LIN {X 0,Y 516.88,Z 308.725,A -85,B 0,C 180,E1 -5018.462,E2 -5018.462} C_VEL
LIN {X 0,Y 516.899,Z 308.722,A -85,B 0,C 180,E1 -5020.954,E2 -5020.954} C_VEL
LIN {X 0,Y 516.911,Z 308.717,A -85,B 0,C 180,E1 -5023.41,E2 -5023.41} C_VEL
LIN {X 0,Y 516.889,Z 308.719,A -85,B 0,C 180,E1 -5025.833,E2 -5025.833} C_VEL
LIN {X 0,Y 516.958,Z 308.715,A -85,B 0,C 180,E1 -5028.233,E2 -5028.233} C_VEL
LIN {X 0,Y 516.963,Z 308.71,A -85,B 0,C 180,E1 -5031.399,E2 -5031.399} C_VEL
LIN {X 0,Y 517.004,Z 308.705,A -85,B 0,C 180,E1 -5033.757,E2 -5033.757} C_VEL
LIN {X 0,Y 517.078,Z 308.696,A -85,B 0,C 180,E1 -5037.663,E2 -5037.663} C_VEL
LIN {X 0,Y 517.088,Z 308.697,A -85,B 0,C 180,E1 -5040.779,E2 -5040.779} C_VEL
LIN {X 0,Y 517.009,Z 308.704,A -85,B 0,C 180,E1 -5043.117,E2 -5043.117} C_VEL
LIN {X 0,Y 517.003,Z 308.713,A -85,B 0,C 180,E1 -5046.243,E2 -5046.243} C_VEL
LIN {X 0,Y 516.948,Z 308.712,A -85,B 0,C 180,E1 -5049.389,E2 -5049.389} C_VEL
LIN {X 0,Y 516.975,Z 308.712,A -85,B 0,C 180,E1 -5051.824,E2 -5051.824} C_VEL
LIN {X 0,Y 516.936,Z 308.713,A -85,B 0,C 180,E1 -5055.147,E2 -5055.147} C_VEL
LIN {X 0,Y 516.918,Z 308.723,A -85,B 0,C 180,E1 -5058.222,E2 -5058.222} C_VEL
LIN {X 0,Y 516.904,Z 308.718,A -85,B 0,C 180,E1 -5060.702,E2 -5060.702} C_VEL
LIN {X 0,Y 516.904,Z 308.726,A -85,B 0,C 180,E1 -5064.072,E2 -5064.072} C_VEL
LIN {X 0,Y 516.919,Z 308.716,A -85,B 0,C 180,E1 -5066.658,E2 -5066.658} C_VEL
LIN {X 0,Y 516.918,Z 308.719,A -85,B 0,C 180,E1 -5069.527,E2 -5069.527} C_VEL
LIN {X 0,Y 516.894,Z 308.719,A -85,B 0,C 180,E1 -5072.545,E2 -5072.545} C_VEL
LIN {X 0,Y 516.877,Z 308.723,A -85,B 0,C 180,E1 -5075.333,E2 -5075.333} C_VEL
LIN {X 0,Y 516.876,Z 308.729,A -85,B 0,C 180,E1 -5077.944,E2 -5077.944} C_VEL
LIN {X 0,Y 516.898,Z 308.72,A -85,B 0,C 180,E1 -5080.74,E2 -5080.74} C_VEL
LIN {X 0,Y 516.876,Z 308.729,A -85,B 0,C 180,E1 -5083.904,E2 -5083.904} C_VEL
LIN {X 0,Y 516.878,Z 308.728,A -85,B 0,C 180,E1 -5086.107,E2 -5086.107} C_VEL
LIN {X 0,Y 516.909,Z 308.84,A -85,B 0,C 180,E1 -5087.678,E2 -5087.678} C_VEL
LIN {X 0,Y 519.073,Z 319.078,A -85,B 0,C 180,E1 -5090.481,E2 -5090.481} C_VEL
LIN {X 0,Y 519.423,Z 323.098,A -85,B 0,C 180,E1 -5091.51,E2 -5091.51} C_VEL
LIN {X 0,Y 518.871,Z 335.018,A -85,B 0,C 180,E1 -5094.38,E2 -5094.38} C_VEL
LIN {X 0,Y 518.422,Z 347.059,A -85,B 0,C 180,E1 -5097.193,E2 -5097.193} C_VEL
LIN {X 0,Y 518.122,Z 360.493,A -85,B 0,C 180,E1 -5100.241,E2 -5100.241} C_VEL
LIN {X 0,Y 517.829,Z 372.841,A -85,B 0,C 180,E1 -5102.958,E2 -5102.958} C_VEL
LIN {X 0,Y 517.584,Z 386.839,A -85,B 0,C 180,E1 -5105.962,E2 -5105.962} C_VEL
LIN {X 0,Y 517.289,Z 401.876,A -85,B 0,C 180,E1 -5109.107,E2 -5109.107} C_VEL
LIN {X 0,Y 517.084,Z 414.888,A -85,B 0,C 180,E1 -5111.784,E2 -5111.784} C_VEL
LIN {X 0,Y 516.986,Z 421.677,A -85,B 0,C 180,E1 -5113.134,E2 -5113.134} C_VEL
LIN {X 0,Y 517.227,Z 423.856,A -85,B 0,C 180,E1 -5113.225,E2 -5113.225} C_VEL
LIN {X 0,Y 519.477,Z 437.499,A -85,B 0,C 180,E1 -5113.56,E2 -5113.56} C_VEL
LIN {X 0,Y 519.127,Z 450.989,A -85,B 0,C 180,E1 -5113.956,E2 -5113.956} C_VEL
LIN {X 0,Y 518.793,Z 464.997,A -85,B 0,C 180,E1 -5114.533,E2 -5114.533} C_VEL
LIN {X 0,Y 518.401,Z 478.733,A -85,B 0,C 180,E1 -5115.275,E2 -5115.275} C_VEL
LIN {X 0,Y 517.975,Z 491.802,A -85,B 0,C 180,E1 -5116.165,E2 -5116.165} C_VEL
LIN {X 0,Y 517.58,Z 503.611,A -85,B 0,C 180,E1 -5117.154,E2 -5117.154} C_VEL
LIN {X 0,Y 517.291,Z 514.343,A -85,B 0,C 180,E1 -5118.242,E2 -5118.242} C_VEL
LIN {X 0,Y 516.97,Z 524.044,A -85,B 0,C 180,E1 -5119.426,E2 -5119.426} C_VEL
LIN {X 0,Y 516.703,Z 533.314,A -85,B 0,C 180,E1 -5120.804,E2 -5120.804} C_VEL
LIN {X 0,Y 516.5,Z 540.804,A -85,B 0,C 180,E1 -5122.18,E2 -5122.18} C_VEL
LIN {X 0,Y 516.449,Z 546.275,A -85,B 0,C 180,E1 -5123.418,E2 -5123.418} C_VEL
LIN {X 0,Y 516.387,Z 550.181,A -85,B 0,C 180,E1 -5124.534,E2 -5124.534} C_VEL
LIN {X 0,Y 516.324,Z 554.317,A -85,B 0,C 180,E1 -5126.098,E2 -5126.098} C_VEL
LIN {X 0,Y 516.259,Z 557.003,A -85,B 0,C 180,E1 -5127.66,E2 -5127.66} C_VEL
LIN {X 0,Y 516.157,Z 558.334,A -85,B 0,C 180,E1 -5129.221,E2 -5129.221} C_VEL
LIN {X 0,Y 516.157,Z 558.334,A -85,B 0,C 180,E1 -5130.781,E2 -5130.781} C_VEL
LIN {X 0,Y 516.26,Z 557.004,A -85,B 0,C 180,E1 -5132.341,E2 -5132.341} C_VEL
LIN {X 0,Y 516.325,Z 554.318,A -85,B 0,C 180,E1 -5133.903,E2 -5133.903} C_VEL
LIN {X 0,Y 516.388,Z 550.177,A -85,B 0,C 180,E1 -5135.467,E2 -5135.467} C_VEL
LIN {X 0,Y 516.42,Z 545.4,A -85,B 0,C 180,E1 -5136.795,E2 -5136.795} C_VEL
LIN {X 0,Y 516.576,Z 538.799,A -85,B 0,C 180,E1 -5138.214,E2 -5138.214} C_VEL
LIN {X 0,Y 516.766,Z 530.746,A -85,B 0,C 180,E1 -5139.591,E2 -5139.591} C_VEL
LIN {X 0,Y 517.019,Z 522.341,A -85,B 0,C 180,E1 -5140.773,E2 -5140.773} C_VEL
LIN {X 0,Y 517.337,Z 511.736,A -85,B 0,C 180,E1 -5142.008,E2 -5142.008} C_VEL
LIN {X 0,Y 517.627,Z 500.961,A -85,B 0,C 180,E1 -5143.046,E2 -5143.046} C_VEL
LIN {X 0,Y 518.02,Z 488.509,A -85,B 0,C 180,E1 -5144.035,E2 -5144.035} C_VEL
LIN {X 0,Y 518.462,Z 476.278,A -85,B 0,C 180,E1 -5144.825,E2 -5144.825} C_VEL
LIN {X 0,Y 518.779,Z 462.835,A -85,B 0,C 180,E1 -5145.52,E2 -5145.52} C_VEL
LIN {X 0,Y 519.088,Z 448.451,A -85,B 0,C 180,E1 -5146.084,E2 -5146.084} C_VEL
LIN {X 0,Y 519.278,Z 435.91,A -85,B 0,C 180,E1 -5146.444,E2 -5146.444} C_VEL
LIN {X 0,Y 517.254,Z 424.028,A -85,B 0,C 180,E1 -5146.737,E2 -5146.737} C_VEL
LIN {X 0,Y 516.973,Z 420.832,A -85,B 0,C 180,E1 -5146.817,E2 -5146.817} C_VEL
LIN {X 0,Y 516.989,Z 419.507,A -85,B 0,C 180,E1 -5146.995,E2 -5146.995} C_VEL
LIN {X 0,Y 517.158,Z 403.396,A -85,B 0,C 180,E1 -5150.096,E2 -5150.096} C_VEL
LIN {X 0,Y 517.275,Z 387.291,A -85,B 0,C 180,E1 -5153.205,E2 -5153.205} C_VEL
LIN {X 0,Y 517.316,Z 371.528,A -85,B 0,C 180,E1 -5156.28,E2 -5156.28} C_VEL
LIN {X 0,Y 517.349,Z 356.477,A -85,B 0,C 180,E1 -5159.279,E2 -5159.279} C_VEL
LIN {X 0,Y 517.299,Z 343.291,A -85,B 0,C 180,E1 -5161.996,E2 -5161.996} C_VEL
LIN {X 0,Y 517.529,Z 327.436,A -85,B 0,C 180,E1 -5165.433,E2 -5165.433} C_VEL
LIN {X 0,Y 518.077,Z 316.945,A -85,B 0,C 180,E1 -5167.87,E2 -5167.87} C_VEL
LIN {X 0,Y 517.489,Z 311.544,A -85,B 0,C 180,E1 -5169.275,E2 -5169.275} C_VEL
LIN {X 0,Y 516.91,Z 308.795,A -85,B 0,C 180,E1 -5170.095,E2 -5170.095} C_VEL
LIN {X 0,Y 516.908,Z 308.721,A -85,B 0,C 180,E1 -5172.829,E2 -5172.829} C_VEL
LIN {X 0,Y 516.926,Z 308.72,A -85,B 0,C 180,E1 -5175.01,E2 -5175.01} C_VEL
LIN {X 0,Y 516.926,Z 308.718,A -85,B 0,C 180,E1 -5178.398,E2 -5178.398} C_VEL
LIN {X 0,Y 516.89,Z 308.726,A -85,B 0,C 180,E1 -5181.285,E2 -5181.285} C_VEL
LIN {X 0,Y 516.896,Z 308.72,A -85,B 0,C 180,E1 -5184.222,E2 -5184.222} C_VEL
LIN {X 0,Y 516.899,Z 308.724,A -85,B 0,C 180,E1 -5187.053,E2 -5187.053} C_VEL
LIN {X 0,Y 516.895,Z 308.723,A -85,B 0,C 180,E1 -5189.797,E2 -5189.797} C_VEL
LIN {X 0,Y 516.932,Z 308.716,A -85,B 0,C 180,E1 -5192.468,E2 -5192.468} C_VEL
LIN {X 0,Y 516.914,Z 308.724,A -85,B 0,C 180,E1 -5195.072,E2 -5195.072} C_VEL
LIN {X 0,Y 516.873,Z 308.729,A -85,B 0,C 180,E1 -5197.622,E2 -5197.622} C_VEL
LIN {X 0,Y 516.936,Z 308.718,A -85,B 0,C 180,E1 -5200.13,E2 -5200.13} C_VEL
LIN {X 0,Y 516.965,Z 308.871,A -85,B 0,C 180,E1 -5202.929,E2 -5202.929} C_VEL
LIN {X 0,Y 517.172,Z 309.892,A -85,B 0,C 180,E1 -5203.063,E2 -5203.063} C_VEL
LIN {X 0,Y 519.287,Z 316.798,A -85,B 0,C 180,E1 -5203.438,E2 -5203.438} C_VEL
LIN {X 0,Y 518.946,Z 329.14,A -85,B 0,C 180,E1 -5204.059,E2 -5204.059} C_VEL
LIN {X 0,Y 518.599,Z 341.91,A -85,B 0,C 180,E1 -5204.878,E2 -5204.878} C_VEL
LIN {X 0,Y 518.209,Z 353.156,A -85,B 0,C 180,E1 -5205.77,E2 -5205.77} C_VEL
LIN {X 0,Y 517.779,Z 364.396,A -85,B 0,C 180,E1 -5206.859,E2 -5206.859} C_VEL
LIN {X 0,Y 517.422,Z 373.649,A -85,B 0,C 180,E1 -5207.949,E2 -5207.949} C_VEL
LIN {X 0,Y 517.166,Z 382.603,A -85,B 0,C 180,E1 -5209.231,E2 -5209.231} C_VEL
LIN {X 0,Y 516.868,Z 390.417,A -85,B 0,C 180,E1 -5210.609,E2 -5210.609} C_VEL
LIN {X 0,Y 516.71,Z 395.872,A -85,B 0,C 180,E1 -5211.789,E2 -5211.789} C_VEL
LIN {X 0,Y 516.544,Z 401.506,A -85,B 0,C 180,E1 -5213.329,E2 -5213.329} C_VEL
LIN {X 0,Y 516.491,Z 404.86,A -85,B 0,C 180,E1 -5214.534,E2 -5214.534} C_VEL
LIN {X 0,Y 516.418,Z 407.939,A -85,B 0,C 180,E1 -5216.098,E2 -5216.098} C_VEL
LIN {X 0,Y 516.325,Z 409.711,A -85,B 0,C 180,E1 -5217.66,E2 -5217.66} C_VEL
LIN {X 0,Y 516.262,Z 410.169,A -85,B 0,C 180,E1 -5219.22,E2 -5219.22} C_VEL
LIN {X 0,Y 516.266,Z 409.359,A -85,B 0,C 180,E1 -5220.78,E2 -5220.78} C_VEL
LIN {X 0,Y 516.334,Z 407.231,A -85,B 0,C 180,E1 -5222.34,E2 -5222.34} C_VEL
LIN {X 0,Y 516.478,Z 403.747,A -85,B 0,C 180,E1 -5223.902,E2 -5223.902} C_VEL
LIN {X 0,Y 516.523,Z 398.812,A -85,B 0,C 180,E1 -5225.466,E2 -5225.466} C_VEL
LIN {X 0,Y 516.725,Z 392.217,A -85,B 0,C 180,E1 -5227.031,E2 -5227.031} C_VEL
LIN {X 0,Y 516.936,Z 384.86,A -85,B 0,C 180,E1 -5228.404,E2 -5228.404} C_VEL
LIN {X 0,Y 517.244,Z 375.735,A -85,B 0,C 180,E1 -5229.779,E2 -5229.779} C_VEL
LIN {X 0,Y 517.558,Z 366.136,A -85,B 0,C 180,E1 -5230.959,E2 -5230.959} C_VEL
LIN {X 0,Y 517.969,Z 355.356,A -85,B 0,C 180,E1 -5232.053,E2 -5232.053} C_VEL
LIN {X 0,Y 518.386,Z 343.631,A -85,B 0,C 180,E1 -5233.026,E2 -5233.026} C_VEL
LIN {X 0,Y 518.76,Z 331.962,A -85,B 0,C 180,E1 -5233.815,E2 -5233.815} C_VEL
LIN {X 0,Y 519.118,Z 319.213,A -85,B 0,C 180,E1 -5234.505,E2 -5234.505} C_VEL
LIN {X 0,Y 519.013,Z 315.975,A -85,B 0,C 180,E1 -5234.658,E2 -5234.658} C_VEL
LIN {X 0,Y 517.066,Z 309.275,A -85,B 0,C 180,E1 -5235.044,E2 -5235.044} C_VEL
LIN {X 0,Y 516.959,Z 308.748,A -85,B 0,C 180,E1 -5235.195,E2 -5235.195} C_VEL
LIN {X 0,Y 516.93,Z 308.718,A -85,B 0,C 180,E1 -5238.222,E2 -5238.222} C_VEL
LIN {X 0,Y 516.917,Z 308.724,A -85,B 0,C 180,E1 -5240.702,E2 -5240.702} C_VEL
LIN {X 0,Y 516.908,Z 308.719,A -85,B 0,C 180,E1 -5244.072,E2 -5244.072} C_VEL
LIN {X 0,Y 516.929,Z 308.723,A -85,B 0,C 180,E1 -5246.658,E2 -5246.658} C_VEL
LIN {X 0,Y 516.916,Z 308.716,A -85,B 0,C 180,E1 -5249.524,E2 -5249.524} C_VEL
LIN {X 0,Y 516.9,Z 308.726,A -85,B 0,C 180,E1 -5252.543,E2 -5252.543} C_VEL
LIN {X 0,Y 516.885,Z 308.72,A -85,B 0,C 180,E1 -5255.332,E2 -5255.332} C_VEL
LIN {X 0,Y 516.886,Z 308.721,A -85,B 0,C 180,E1 -5257.943,E2 -5257.943} C_VEL
LIN {X 0,Y 516.888,Z 308.724,A -85,B 0,C 180,E1 -5260.742,E2 -5260.742} C_VEL
LIN {X 0,Y 516.888,Z 308.723,A -85,B 0,C 180,E1 -5262.832,E2 -5262.832} C_VEL
LIN {X 0,Y 516.898,Z 308.718,A -85,B 0,C 180,E1 -5265.323,E2 -5265.323} C_VEL
LIN {X 0,Y 516.211,Z 308.807,A -85,B 0,C 180,E1 -5265.974,E2 -5265.974} C_VEL
LIN {X 0,Y 513.372,Z 309.164,A -85,B 0,C 180,E1 -5267.03,E2 -5267.03} C_VEL
LIN {X 0,Y 510.978,Z 309.464,A -85,B 0,C 180,E1 -5267.881,E2 -5267.881} C_VEL
LIN {X 0,Y 509.941,Z 309.591,A -85,B 0,C 180,E1 -5268.538,E2 -5268.538} C_VEL
LIN {X 0,Y 509.851,Z 309.599,A -85,B 0,C 180,E1 -5268.761,E2 -5268.761} C_VEL
LIN {X 0,Y 509.856,Z 309.597,A -85,B 0,C 180,E1 -5271.786,E2 -5271.786} C_VEL
LIN {X 0,Y 509.836,Z 309.602,A -85,B 0,C 180,E1 -5274.622,E2 -5274.622} C_VEL
LIN {X 0,Y 509.867,Z 309.594,A -85,B 0,C 180,E1 -5277.481,E2 -5277.481} C_VEL
LIN {X 0,Y 509.865,Z 309.602,A -85,B 0,C 180,E1 -5280.273,E2 -5280.273} C_VEL
LIN {X 0,Y 509.892,Z 309.591,A -85,B 0,C 180,E1 -5282.944,E2 -5282.944} C_VEL
LIN {X 0,Y 509.858,Z 309.597,A -85,B 0,C 180,E1 -5285.573,E2 -5285.573} C_VEL
LIN {X 0,Y 509.829,Z 309.606,A -85,B 0,C 180,E1 -5288.148,E2 -5288.148} C_VEL
LIN {X 0,Y 509.87,Z 309.594,A -85,B 0,C 180,E1 -5290.681,E2 -5290.681} C_VEL
LIN {X 0,Y 509.891,Z 309.591,A -85,B 0,C 180,E1 -5293.174,E2 -5293.174} C_VEL
LIN {X 0,Y 509.871,Z 309.597,A -85,B 0,C 180,E1 -5295.634,E2 -5295.634} C_VEL
LIN {X 0,Y 509.92,Z 309.587,A -85,B 0,C 180,E1 -5298.874,E2 -5298.874} C_VEL
LIN {X 0,Y 509.957,Z 309.588,A -85,B 0,C 180,E1 -5302.078,E2 -5302.078} C_VEL
LIN {X 0,Y 509.985,Z 309.58,A -85,B 0,C 180,E1 -5304.464,E2 -5304.464} C_VEL
LIN {X 0,Y 510.061,Z 309.576,A -85,B 0,C 180,E1 -5307.63,E2 -5307.63} C_VEL
LIN {X 0,Y 510.069,Z 309.569,A -85,B 0,C 180,E1 -5310.789,E2 -5310.789} C_VEL
LIN {X 0,Y 509.959,Z 309.584,A -85,B 0,C 180,E1 -5313.159,E2 -5313.159} C_VEL
LIN {X 0,Y 509.984,Z 309.58,A -85,B 0,C 180,E1 -5316.329,E2 -5316.329} C_VEL
LIN {X 0,Y 509.919,Z 309.587,A -85,B 0,C 180,E1 -5318.719,E2 -5318.719} C_VEL
LIN {X 0,Y 509.908,Z 309.592,A -85,B 0,C 180,E1 -5321.931,E2 -5321.931} C_VEL
LIN {X 0,Y 509.897,Z 309.595,A -85,B 0,C 180,E1 -5325.241,E2 -5325.241} C_VEL
LIN {X 0,Y 509.892,Z 309.593,A -85,B 0,C 180,E1 -5328,E2 -5328} C_VEL
LIN {X 0,Y 509.853,Z 309.598,A -85,B 0,C 180,E1 -5331.001,E2 -5331.001} C_VEL
LIN {X 0,Y 509.839,Z 309.603,A -85,B 0,C 180,E1 -5333.562,E2 -5333.562} C_VEL
LIN {X 0,Y 509.913,Z 309.588,A -85,B 0,C 180,E1 -5336.378,E2 -5336.378} C_VEL
LIN {X 0,Y 509.877,Z 309.595,A -85,B 0,C 180,E1 -5338.843,E2 -5338.843} C_VEL
LIN {X 0,Y 509.826,Z 309.603,A -85,B 0,C 180,E1 -5341.589,E2 -5341.589} C_VEL
LIN {X 0,Y 509.85,Z 309.596,A -85,B 0,C 180,E1 -5344.412,E2 -5344.412} C_VEL
LIN {X 0,Y 509.815,Z 309.607,A -85,B 0,C 180,E1 -5347.34,E2 -5347.34} C_VEL
LIN {X 0,Y 509.837,Z 309.598,A -85,B 0,C 180,E1 -5350.381,E2 -5350.381} C_VEL
LIN {X 0,Y 509.838,Z 309.606,A -85,B 0,C 180,E1 -5353.063,E2 -5353.063} C_VEL
LIN {X 0,Y 509.827,Z 309.599,A -85,B 0,C 180,E1 -5355.791,E2 -5355.791} C_VEL
LIN {X 0,Y 509.855,Z 309.598,A -85,B 0,C 180,E1 -5358.574,E2 -5358.574} C_VEL
LIN {X 0,Y 509.848,Z 309.596,A -85,B 0,C 180,E1 -5361.785,E2 -5361.785} C_VEL
LIN {X 0,Y 509.842,Z 309.601,A -85,B 0,C 180,E1 -5364.622,E2 -5364.622} C_VEL
LIN {X 0,Y 509.861,Z 309.596,A -85,B 0,C 180,E1 -5367.48,E2 -5367.48} C_VEL
LIN {X 0,Y 509.876,Z 309.594,A -85,B 0,C 180,E1 -5370.268,E2 -5370.268} C_VEL
LIN {X 0,Y 509.882,Z 309.598,A -85,B 0,C 180,E1 -5372.944,E2 -5372.944} C_VEL
LIN {X 0,Y 509.864,Z 309.594,A -85,B 0,C 180,E1 -5375.573,E2 -5375.573} C_VEL
LIN {X 0,Y 509.816,Z 309.602,A -85,B 0,C 180,E1 -5378.148,E2 -5378.148} C_VEL
LIN {X 0,Y 509.859,Z 309.604,A -85,B 0,C 180,E1 -5380.681,E2 -5380.681} C_VEL
LIN {X 0,Y 509.881,Z 309.594,A -85,B 0,C 180,E1 -5383.174,E2 -5383.174} C_VEL
LIN {X 0,Y 509.857,Z 309.595,A -85,B 0,C 180,E1 -5385.634,E2 -5385.634} C_VEL
LIN {X 0,Y 509.906,Z 309.593,A -85,B 0,C 180,E1 -5388.874,E2 -5388.874} C_VEL
LIN {X 0,Y 509.944,Z 309.587,A -85,B 0,C 180,E1 -5392.078,E2 -5392.078} C_VEL
LIN {X 0,Y 509.977,Z 309.589,A -85,B 0,C 180,E1 -5394.464,E2 -5394.464} C_VEL
LIN {X 0,Y 510.048,Z 309.571,A -85,B 0,C 180,E1 -5397.631,E2 -5397.631} C_VEL
LIN {X 0,Y 510.058,Z 309.573,A -85,B 0,C 180,E1 -5400.789,E2 -5400.789} C_VEL
LIN {X 0,Y 509.951,Z 309.583,A -85,B 0,C 180,E1 -5403.16,E2 -5403.16} C_VEL
LIN {X 0,Y 509.971,Z 309.589,A -85,B 0,C 180,E1 -5406.33,E2 -5406.33} C_VEL
LIN {X 0,Y 509.909,Z 309.591,A -85,B 0,C 180,E1 -5408.72,E2 -5408.72} C_VEL
LIN {X 0,Y 509.943,Z 309.589,A -85,B 0,C 180,E1 -5411.931,E2 -5411.931} C_VEL
LIN {X 0,Y 509.885,Z 309.591,A -85,B 0,C 180,E1 -5415.242,E2 -5415.242} C_VEL
LIN {X 0,Y 509.881,Z 309.599,A -85,B 0,C 180,E1 -5418.001,E2 -5418.001} C_VEL
LIN {X 0,Y 509.842,Z 309.597,A -85,B 0,C 180,E1 -5421.002,E2 -5421.002} C_VEL
LIN {X 0,Y 509.829,Z 309.601,A -85,B 0,C 180,E1 -5423.563,E2 -5423.563} C_VEL
LIN {X 0,Y 509.904,Z 309.592,A -85,B 0,C 180,E1 -5426.379,E2 -5426.379} C_VEL
LIN {X 0,Y 509.878,Z 309.592,A -85,B 0,C 180,E1 -5428.844,E2 -5428.844} C_VEL
LIN {X 0,Y 509.82,Z 309.604,A -85,B 0,C 180,E1 -5431.59,E2 -5431.59} C_VEL
LIN {X 0,Y 509.847,Z 309.598,A -85,B 0,C 180,E1 -5434.414,E2 -5434.414} C_VEL
LIN {X 0,Y 509.813,Z 309.605,A -85,B 0,C 180,E1 -5437.341,E2 -5437.341} C_VEL
LIN {X 0,Y 509.856,Z 309.599,A -85,B 0,C 180,E1 -5440.381,E2 -5440.381} C_VEL
LIN {X 0,Y 509.818,Z 309.605,A -85,B 0,C 180,E1 -5443.063,E2 -5443.063} C_VEL
LIN {X 0,Y 509.826,Z 309.608,A -85,B 0,C 180,E1 -5445.793,E2 -5445.793} C_VEL
LIN {X 0,Y 509.881,Z 309.828,A -85,B 0,C 180,E1 -5447.4,E2 -5447.4} C_VEL
LIN {X 0,Y 511.687,Z 318.431,A -85,B 0,C 180,E1 -5449.795,E2 -5449.795} C_VEL
LIN {X 0,Y 512.527,Z 323.727,A -85,B 0,C 180,E1 -5451.202,E2 -5451.202} C_VEL
LIN {X 0,Y 512.044,Z 334.436,A -85,B 0,C 180,E1 -5453.831,E2 -5453.831} C_VEL
LIN {X 0,Y 511.507,Z 347.536,A -85,B 0,C 180,E1 -5456.943,E2 -5456.943} C_VEL
LIN {X 0,Y 511.149,Z 360.882,A -85,B 0,C 180,E1 -5460.021,E2 -5460.021} C_VEL
LIN {X 0,Y 510.847,Z 372.194,A -85,B 0,C 180,E1 -5462.557,E2 -5462.557} C_VEL
LIN {X 0,Y 510.544,Z 386.148,A -85,B 0,C 180,E1 -5465.609,E2 -5465.609} C_VEL
LIN {X 0,Y 510.296,Z 398.128,A -85,B 0,C 180,E1 -5468.171,E2 -5468.171} C_VEL
LIN {X 0,Y 510.092,Z 410.122,A -85,B 0,C 180,E1 -5470.691,E2 -5470.691} C_VEL
LIN {X 0,Y 509.941,Z 420.851,A -85,B 0,C 180,E1 -5472.894,E2 -5472.894} C_VEL
LIN {X 0,Y 510.193,Z 423.351,A -85,B 0,C 180,E1 -5472.998,E2 -5472.998} C_VEL
LIN {X 0,Y 512.36,Z 436.055,A -85,B 0,C 180,E1 -5473.319,E2 -5473.319} C_VEL
LIN {X 0,Y 512.48,Z 441.801,A -85,B 0,C 180,E1 -5473.479,E2 -5473.479} C_VEL
LIN {X 0,Y 512.122,Z 455.944,A -85,B 0,C 180,E1 -5473.968,E2 -5473.968} C_VEL
LIN {X 0,Y 511.75,Z 468.895,A -85,B 0,C 180,E1 -5474.57,E2 -5474.57} C_VEL
LIN {X 0,Y 511.276,Z 482.375,A -85,B 0,C 180,E1 -5475.37,E2 -5475.37} C_VEL
LIN {X 0,Y 510.885,Z 494.554,A -85,B 0,C 180,E1 -5476.274,E2 -5476.274} C_VEL
LIN {X 0,Y 510.443,Z 505.691,A -85,B 0,C 180,E1 -5477.274,E2 -5477.274} C_VEL
LIN {X 0,Y 510.154,Z 516.735,A -85,B 0,C 180,E1 -5478.478,E2 -5478.478} C_VEL
LIN {X 0,Y 509.802,Z 525.854,A -85,B 0,C 180,E1 -5479.677,E2 -5479.677} C_VEL
LIN {X 0,Y 509.579,Z 534.617,A -85,B 0,C 180,E1 -5481.075,E2 -5481.075} C_VEL
LIN {X 0,Y 509.389,Z 541.684,A -85,B 0,C 180,E1 -5482.469,E2 -5482.469} C_VEL
LIN {X 0,Y 509.334,Z 546.571,A -85,B 0,C 180,E1 -5483.663,E2 -5483.663} C_VEL
LIN {X 0,Y 509.247,Z 550.523,A -85,B 0,C 180,E1 -5484.854,E2 -5484.854} C_VEL
LIN {X 0,Y 509.252,Z 553.577,A -85,B 0,C 180,E1 -5486.044,E2 -5486.044} C_VEL
LIN {X 0,Y 509.188,Z 556.364,A -85,B 0,C 180,E1 -5487.628,E2 -5487.628} C_VEL
LIN {X 0,Y 509.083,Z 557.731,A -85,B 0,C 180,E1 -5489.21,E2 -5489.21} C_VEL
LIN {X 0,Y 509.083,Z 557.724,A -85,B 0,C 180,E1 -5490.792,E2 -5490.792} C_VEL
LIN {X 0,Y 509.188,Z 556.341,A -85,B 0,C 180,E1 -5492.374,E2 -5492.374} C_VEL
LIN {X 0,Y 509.253,Z 553.531,A -85,B 0,C 180,E1 -5493.957,E2 -5493.957} C_VEL
LIN {X 0,Y 509.323,Z 549.216,A -85,B 0,C 180,E1 -5495.544,E2 -5495.544} C_VEL
LIN {X 0,Y 509.352,Z 544.436,A -85,B 0,C 180,E1 -5496.855,E2 -5496.855} C_VEL
LIN {X 0,Y 509.526,Z 537.6,A -85,B 0,C 180,E1 -5498.328,E2 -5498.328} C_VEL
LIN {X 0,Y 509.702,Z 529.49,A -85,B 0,C 180,E1 -5499.725,E2 -5499.725} C_VEL
LIN {X 0,Y 509.951,Z 521.024,A -85,B 0,C 180,E1 -5500.924,E2 -5500.924} C_VEL
LIN {X 0,Y 510.282,Z 510.37,A -85,B 0,C 180,E1 -5502.175,E2 -5502.175} C_VEL
LIN {X 0,Y 510.61,Z 499.506,A -85,B 0,C 180,E1 -5503.229,E2 -5503.229} C_VEL
LIN {X 0,Y 511.013,Z 486.978,A -85,B 0,C 180,E1 -5504.232,E2 -5504.232} C_VEL
LIN {X 0,Y 511.457,Z 474.662,A -85,B 0,C 180,E1 -5505.033,E2 -5505.033} C_VEL
LIN {X 0,Y 511.873,Z 461.127,A -85,B 0,C 180,E1 -5505.734,E2 -5505.734} C_VEL
LIN {X 0,Y 512.217,Z 446.813,A -85,B 0,C 180,E1 -5506.3,E2 -5506.3} C_VEL
LIN {X 0,Y 512.3,Z 436.585,A -85,B 0,C 180,E1 -5506.611,E2 -5506.611} C_VEL
LIN {X 0,Y 510.437,Z 425.239,A -85,B 0,C 180,E1 -5506.91,E2 -5506.91} C_VEL
LIN {X 0,Y 509.897,Z 419.326,A -85,B 0,C 180,E1 -5507.058,E2 -5507.058} C_VEL
LIN {X 0,Y 509.903,Z 417.037,A -85,B 0,C 180,E1 -5507.445,E2 -5507.445} C_VEL
LIN {X 0,Y 510.075,Z 401.604,A -85,B 0,C 180,E1 -5510.458,E2 -5510.458} C_VEL
LIN {X 0,Y 510.213,Z 385.864,A -85,B 0,C 180,E1 -5513.545,E2 -5513.545} C_VEL
LIN {X 0,Y 510.25,Z 371.225,A -85,B 0,C 180,E1 -5516.455,E2 -5516.455} C_VEL
LIN {X 0,Y 510.294,Z 357.373,A -85,B 0,C 180,E1 -5519.27,E2 -5519.27} C_VEL
LIN {X 0,Y 510.277,Z 344.266,A -85,B 0,C 180,E1 -5522.023,E2 -5522.023} C_VEL
LIN {X 0,Y 510.585,Z 327.718,A -85,B 0,C 180,E1 -5525.697,E2 -5525.697} C_VEL
LIN {X 0,Y 511.106,Z 319.175,A -85,B 0,C 180,E1 -5527.728,E2 -5527.728} C_VEL
LIN {X 0,Y 510.94,Z 315.102,A -85,B 0,C 180,E1 -5528.778,E2 -5528.778} C_VEL
LIN {X 0,Y 509.854,Z 309.671,A -85,B 0,C 180,E1 -5530.381,E2 -5530.381} C_VEL
LIN {X 0,Y 509.843,Z 309.603,A -85,B 0,C 180,E1 -5533.065,E2 -5533.065} C_VEL
LIN {X 0,Y 509.834,Z 309.606,A -85,B 0,C 180,E1 -5535.793,E2 -5535.793} C_VEL
LIN {X 0,Y 509.869,Z 309.597,A -85,B 0,C 180,E1 -5538.576,E2 -5538.576} C_VEL
LIN {X 0,Y 509.856,Z 309.602,A -85,B 0,C 180,E1 -5541.786,E2 -5541.786} C_VEL
LIN {X 0,Y 509.85,Z 309.598,A -85,B 0,C 180,E1 -5544.624,E2 -5544.624} C_VEL
LIN {X 0,Y 509.866,Z 309.602,A -85,B 0,C 180,E1 -5547.481,E2 -5547.481} C_VEL
LIN {X 0,Y 509.862,Z 309.596,A -85,B 0,C 180,E1 -5550.274,E2 -5550.274} C_VEL
LIN {X 0,Y 509.889,Z 309.597,A -85,B 0,C 180,E1 -5552.945,E2 -5552.945} C_VEL
LIN {X 0,Y 509.873,Z 309.6,A -85,B 0,C 180,E1 -5555.574,E2 -5555.574} C_VEL
LIN {X 0,Y 509.826,Z 309.603,A -85,B 0,C 180,E1 -5558.149,E2 -5558.149} C_VEL
LIN {X 0,Y 509.868,Z 309.601,A -85,B 0,C 180,E1 -5560.682,E2 -5560.682} C_VEL
LIN {X 0,Y 509.929,Z 309.794,A -85,B 0,C 180,E1 -5562.712,E2 -5562.712} C_VEL
LIN {X 0,Y 510.185,Z 310.922,A -85,B 0,C 180,E1 -5562.85,E2 -5562.85} C_VEL
LIN {X 0,Y 512.472,Z 318.387,A -85,B 0,C 180,E1 -5563.262,E2 -5563.262} C_VEL
LIN {X 0,Y 512.087,Z 331.832,A -85,B 0,C 180,E1 -5563.963,E2 -5563.963} C_VEL
LIN {X 0,Y 511.751,Z 344.006,A -85,B 0,C 180,E1 -5564.773,E2 -5564.773} C_VEL
LIN {X 0,Y 511.296,Z 355.084,A -85,B 0,C 180,E1 -5565.675,E2 -5565.675} C_VEL
LIN {X 0,Y 510.924,Z 365.237,A -85,B 0,C 180,E1 -5566.679,E2 -5566.679} C_VEL
LIN {X 0,Y 510.54,Z 374.582,A -85,B 0,C 180,E1 -5567.79,E2 -5567.79} C_VEL
LIN {X 0,Y 510.25,Z 383.546,A -85,B 0,C 180,E1 -5569.083,E2 -5569.083} C_VEL
LIN {X 0,Y 509.924,Z 391.395,A -85,B 0,C 180,E1 -5570.48,E2 -5570.48} C_VEL
LIN {X 0,Y 509.755,Z 396.872,A -85,B 0,C 180,E1 -5571.677,E2 -5571.677} C_VEL
LIN {X 0,Y 509.567,Z 402.505,A -85,B 0,C 180,E1 -5573.234,E2 -5573.234} C_VEL
LIN {X 0,Y 509.495,Z 405.876,A -85,B 0,C 180,E1 -5574.459,E2 -5574.459} C_VEL
LIN {X 0,Y 509.403,Z 408.974,A -85,B 0,C 180,E1 -5576.045,E2 -5576.045} C_VEL
LIN {X 0,Y 509.305,Z 410.741,A -85,B 0,C 180,E1 -5577.628,E2 -5577.628} C_VEL
LIN {X 0,Y 509.248,Z 411.193,A -85,B 0,C 180,E1 -5579.209,E2 -5579.209} C_VEL
LIN {X 0,Y 509.252,Z 410.371,A -85,B 0,C 180,E1 -5580.791,E2 -5580.791} C_VEL
LIN {X 0,Y 509.31,Z 408.223,A -85,B 0,C 180,E1 -5582.373,E2 -5582.373} C_VEL
LIN {X 0,Y 509.462,Z 404.72,A -85,B 0,C 180,E1 -5583.955,E2 -5583.955} C_VEL
LIN {X 0,Y 509.523,Z 399.765,A -85,B 0,C 180,E1 -5585.541,E2 -5585.541} C_VEL
LIN {X 0,Y 509.712,Z 394.18,A -85,B 0,C 180,E1 -5586.902,E2 -5586.902} C_VEL
LIN {X 0,Y 509.959,Z 386.923,A -85,B 0,C 180,E1 -5588.32,E2 -5588.32} C_VEL
LIN {X 0,Y 510.247,Z 378.068,A -85,B 0,C 180,E1 -5589.714,E2 -5589.714} C_VEL
LIN {X 0,Y 510.599,Z 368.757,A -85,B 0,C 180,E1 -5590.91,E2 -5590.91} C_VEL
LIN {X 0,Y 511.081,Z 358.407,A -85,B 0,C 180,E1 -5592.006,E2 -5592.006} C_VEL
LIN {X 0,Y 511.442,Z 347.016,A -85,B 0,C 180,E1 -5593.004,E2 -5593.004} C_VEL
LIN {X 0,Y 511.842,Z 335.906,A -85,B 0,C 180,E1 -5593.803,E2 -5593.803} C_VEL
LIN {X 0,Y 512.211,Z 322.019,A -85,B 0,C 180,E1 -5594.603,E2 -5594.603} C_VEL
LIN {X 0,Y 512.303,Z 317.882,A -85,B 0,C 180,E1 -5594.804,E2 -5594.804} C_VEL
LIN {X 0,Y 510.035,Z 310.259,A -85,B 0,C 180,E1 -5595.247,E2 -5595.247} C_VEL
LIN {X 0,Y 509.892,Z 309.628,A -85,B 0,C 180,E1 -5595.412,E2 -5595.412} C_VEL
LIN {X 0,Y 509.872,Z 309.601,A -85,B 0,C 180,E1 -5598.484,E2 -5598.484} C_VEL
LIN {X 0,Y 509.855,Z 309.603,A -85,B 0,C 180,E1 -5601.002,E2 -5601.002} C_VEL
LIN {X 0,Y 509.869,Z 309.599,A -85,B 0,C 180,E1 -5604.426,E2 -5604.426} C_VEL
LIN {X 0,Y 509.888,Z 309.595,A -85,B 0,C 180,E1 -5607.056,E2 -5607.056} C_VEL
LIN {X 0,Y 509.862,Z 309.594,A -85,B 0,C 180,E1 -5609.751,E2 -5609.751} C_VEL
LIN {X 0,Y 509.878,Z 309.599,A -85,B 0,C 180,E1 -5612.774,E2 -5612.774} C_VEL
LIN {X 0,Y 509.845,Z 309.596,A -85,B 0,C 180,E1 -5615.581,E2 -5615.581} C_VEL
LIN {X 0,Y 509.855,Z 309.601,A -85,B 0,C 180,E1 -5618.338,E2 -5618.338} C_VEL
LIN {X 0,Y 509.86,Z 309.594,A -85,B 0,C 180,E1 -5621.426,E2 -5621.426} C_VEL
LIN {X 0,Y 509.862,Z 309.6,A -85,B 0,C 180,E1 -5624.668,E2 -5624.668} C_VEL
LIN {X 0,Y 509.866,Z 309.599,A -85,B 0,C 180,E1 -5628.103,E2 -5628.103} C_VEL
LIN {X 0,Y 509.851,Z 309.599,A -85,B 0,C 180,E1 -5628.761,E2 -5628.761} C_VEL
LIN {X 0,Y 509.17,Z 309.681,A -85,B 0,C 180,E1 -5629.421,E2 -5629.421} C_VEL
LIN {X 0,Y 506.323,Z 310.042,A -85,B 0,C 180,E1 -5630.492,E2 -5630.492} C_VEL
LIN {X 0,Y 503.918,Z 310.342,A -85,B 0,C 180,E1 -5631.355,E2 -5631.355} C_VEL
LIN {X 0,Y 502.876,Z 310.469,A -85,B 0,C 180,E1 -5632.021,E2 -5632.021} C_VEL
LIN {X 0,Y 502.786,Z 310.479,A -85,B 0,C 180,E1 -5632.247,E2 -5632.247} C_VEL
LIN {X 0,Y 502.806,Z 310.474,A -85,B 0,C 180,E1 -5635.556,E2 -5635.556} C_VEL
LIN {X 0,Y 502.79,Z 310.48,A -85,B 0,C 180,E1 -5637.915,E2 -5637.915} C_VEL
LIN {X 0,Y 502.831,Z 310.472,A -85,B 0,C 180,E1 -5640.712,E2 -5640.712} C_VEL
LIN {X 0,Y 502.869,Z 310.466,A -85,B 0,C 180,E1 -5643.439,E2 -5643.439} C_VEL
LIN {X 0,Y 502.783,Z 310.485,A -85,B 0,C 180,E1 -5646.085,E2 -5646.085} C_VEL
LIN {X 0,Y 502.79,Z 310.477,A -85,B 0,C 180,E1 -5648.689,E2 -5648.689} C_VEL
LIN {X 0,Y 502.836,Z 310.47,A -85,B 0,C 180,E1 -5651.248,E2 -5651.248} C_VEL
LIN {X 0,Y 502.829,Z 310.476,A -85,B 0,C 180,E1 -5653.767,E2 -5653.767} C_VEL
LIN {X 0,Y 502.837,Z 310.474,A -85,B 0,C 180,E1 -5656.254,E2 -5656.254} C_VEL
LIN {X 0,Y 502.884,Z 310.464,A -85,B 0,C 180,E1 -5658.716,E2 -5658.716} C_VEL
LIN {X 0,Y 502.907,Z 310.468,A -85,B 0,C 180,E1 -5661.966,E2 -5661.966} C_VEL
LIN {X 0,Y 502.939,Z 310.458,A -85,B 0,C 180,E1 -5664.386,E2 -5664.386} C_VEL
LIN {X 0,Y 503.031,Z 310.451,A -85,B 0,C 180,E1 -5667.597,E2 -5667.597} C_VEL
LIN {X 0,Y 503.033,Z 310.45,A -85,B 0,C 180,E1 -5669.999,E2 -5669.999} C_VEL
LIN {X 0,Y 503.03,Z 310.446,A -85,B 0,C 180,E1 -5672.401,E2 -5672.401} C_VEL
LIN {X 0,Y 502.933,Z 310.458,A -85,B 0,C 180,E1 -5676.418,E2 -5676.418} C_VEL
LIN {X 0,Y 502.878,Z 310.465,A -85,B 0,C 180,E1 -5678.842,E2 -5678.842} C_VEL
LIN {X 0,Y 502.85,Z 310.47,A -85,B 0,C 180,E1 -5682.101,E2 -5682.101} C_VEL
LIN {X 0,Y 502.852,Z 310.475,A -85,B 0,C 180,E1 -5685.399,E2 -5685.399} C_VEL
LIN {X 0,Y 502.849,Z 310.469,A -85,B 0,C 180,E1 -5688.121,E2 -5688.121} C_VEL
LIN {X 0,Y 502.831,Z 310.47,A -85,B 0,C 180,E1 -5690.535,E2 -5690.535} C_VEL
LIN {X 0,Y 502.799,Z 310.478,A -85,B 0,C 180,E1 -5693.039,E2 -5693.039} C_VEL
LIN {X 0,Y 502.842,Z 310.473,A -85,B 0,C 180,E1 -5695.674,E2 -5695.674} C_VEL
LIN {X 0,Y 502.841,Z 310.469,A -85,B 0,C 180,E1 -5698.372,E2 -5698.372} C_VEL
LIN {X 0,Y 502.797,Z 310.48,A -85,B 0,C 180,E1 -5701.498,E2 -5701.498} C_VEL
LIN {X 0,Y 502.802,Z 310.474,A -85,B 0,C 180,E1 -5704.443,E2 -5704.443} C_VEL
LIN {X 0,Y 502.776,Z 310.486,A -85,B 0,C 180,E1 -5707.177,E2 -5707.177} C_VEL
LIN {X 0,Y 502.787,Z 310.476,A -85,B 0,C 180,E1 -5710.014,E2 -5710.014} C_VEL
LIN {X 0,Y 502.8,Z 310.474,A -85,B 0,C 180,E1 -5712.198,E2 -5712.198} C_VEL
LIN {X 0,Y 502.797,Z 310.477,A -85,B 0,C 180,E1 -5715.467,E2 -5715.467} C_VEL
LIN {X 0,Y 502.817,Z 310.48,A -85,B 0,C 180,E1 -5718.933,E2 -5718.933} C_VEL
LIN {X 0,Y 502.79,Z 310.475,A -85,B 0,C 180,E1 -5722.045,E2 -5722.045} C_VEL
LIN {X 0,Y 502.805,Z 310.48,A -85,B 0,C 180,E1 -5725.034,E2 -5725.034} C_VEL
LIN {X 0,Y 502.783,Z 310.476,A -85,B 0,C 180,E1 -5727.915,E2 -5727.915} C_VEL
LIN {X 0,Y 502.834,Z 310.477,A -85,B 0,C 180,E1 -5730.712,E2 -5730.712} C_VEL
LIN {X 0,Y 502.875,Z 310.466,A -85,B 0,C 180,E1 -5733.434,E2 -5733.434} C_VEL
LIN {X 0,Y 502.786,Z 310.477,A -85,B 0,C 180,E1 -5736.086,E2 -5736.086} C_VEL
LIN {X 0,Y 502.777,Z 310.486,A -85,B 0,C 180,E1 -5738.688,E2 -5738.688} C_VEL
LIN {X 0,Y 502.824,Z 310.473,A -85,B 0,C 180,E1 -5741.248,E2 -5741.248} C_VEL
LIN {X 0,Y 502.817,Z 310.472,A -85,B 0,C 180,E1 -5743.767,E2 -5743.767} C_VEL
LIN {X 0,Y 502.825,Z 310.475,A -85,B 0,C 180,E1 -5746.254,E2 -5746.254} C_VEL
LIN {X 0,Y 502.87,Z 310.472,A -85,B 0,C 180,E1 -5748.716,E2 -5748.716} C_VEL
LIN {X 0,Y 502.894,Z 310.464,A -85,B 0,C 180,E1 -5751.966,E2 -5751.966} C_VEL
LIN {X 0,Y 502.932,Z 310.465,A -85,B 0,C 180,E1 -5754.386,E2 -5754.386} C_VEL
LIN {X 0,Y 503.018,Z 310.447,A -85,B 0,C 180,E1 -5757.598,E2 -5757.598} C_VEL
LIN {X 0,Y 503.019,Z 310.45,A -85,B 0,C 180,E1 -5760,E2 -5760} C_VEL
LIN {X 0,Y 503.018,Z 310.455,A -85,B 0,C 180,E1 -5762.402,E2 -5762.402} C_VEL
LIN {X 0,Y 502.931,Z 310.459,A -85,B 0,C 180,E1 -5765.613,E2 -5765.613} C_VEL
LIN {X 0,Y 502.894,Z 310.468,A -85,B 0,C 180,E1 -5768.033,E2 -5768.033} C_VEL
LIN {X 0,Y 502.885,Z 310.463,A -85,B 0,C 180,E1 -5771.283,E2 -5771.283} C_VEL
LIN {X 0,Y 502.838,Z 310.473,A -85,B 0,C 180,E1 -5774.571,E2 -5774.571} C_VEL
LIN {X 0,Y 502.854,Z 310.473,A -85,B 0,C 180,E1 -5777.907,E2 -5777.907} C_VEL
LIN {X 0,Y 502.82,Z 310.474,A -85,B 0,C 180,E1 -5780.536,E2 -5780.536} C_VEL
LIN {X 0,Y 502.789,Z 310.475,A -85,B 0,C 180,E1 -5783.041,E2 -5783.041} C_VEL
LIN {X 0,Y 502.833,Z 310.474,A -85,B 0,C 180,E1 -5785.676,E2 -5785.676} C_VEL
LIN {X 0,Y 502.835,Z 310.473,A -85,B 0,C 180,E1 -5788.373,E2 -5788.373} C_VEL
LIN {X 0,Y 502.79,Z 310.478,A -85,B 0,C 180,E1 -5791.5,E2 -5791.5} C_VEL
LIN {X 0,Y 502.8,Z 310.476,A -85,B 0,C 180,E1 -5794.445,E2 -5794.445} C_VEL
LIN {X 0,Y 502.775,Z 310.48,A -85,B 0,C 180,E1 -5797.179,E2 -5797.179} C_VEL
LIN {X 0,Y 502.82,Z 310.48,A -85,B 0,C 180,E1 -5800.012,E2 -5800.012} C_VEL
LIN {X 0,Y 502.767,Z 310.484,A -85,B 0,C 180,E1 -5803.232,E2 -5803.232} C_VEL
LIN {X 0,Y 502.785,Z 310.485,A -85,B 0,C 180,E1 -5805.662,E2 -5805.662} C_VEL
LIN {X 0,Y 502.815,Z 310.603,A -85,B 0,C 180,E1 -5807.042,E2 -5807.042} C_VEL
LIN {X 0,Y 504.691,Z 319.547,A -85,B 0,C 180,E1 -5809.577,E2 -5809.577} C_VEL
LIN {X 0,Y 505.639,Z 325.205,A -85,B 0,C 180,E1 -5811.11,E2 -5811.11} C_VEL
LIN {X 0,Y 505.174,Z 335.141,A -85,B 0,C 180,E1 -5813.583,E2 -5813.583} C_VEL
LIN {X 0,Y 504.599,Z 347.998,A -85,B 0,C 180,E1 -5816.686,E2 -5816.686} C_VEL
LIN {X 0,Y 504.213,Z 361.231,A -85,B 0,C 180,E1 -5819.79,E2 -5819.79} C_VEL
LIN {X 0,Y 503.835,Z 373.532,A -85,B 0,C 180,E1 -5822.593,E2 -5822.593} C_VEL
LIN {X 0,Y 503.519,Z 387.452,A -85,B 0,C 180,E1 -5825.686,E2 -5825.686} C_VEL
LIN {X 0,Y 503.22,Z 399.378,A -85,B 0,C 180,E1 -5828.279,E2 -5828.279} C_VEL
LIN {X 0,Y 503.012,Z 411.318,A -85,B 0,C 180,E1 -5830.833,E2 -5830.833} C_VEL
LIN {X 0,Y 502.904,Z 420.242,A -85,B 0,C 180,E1 -5832.673,E2 -5832.673} C_VEL
LIN {X 0,Y 503.499,Z 425.333,A -85,B 0,C 180,E1 -5832.818,E2 -5832.818} C_VEL
LIN {X 0,Y 505.698,Z 439.053,A -85,B 0,C 180,E1 -5833.204,E2 -5833.204} C_VEL
LIN {X 0,Y 505.255,Z 453.612,A -85,B 0,C 180,E1 -5833.694,E2 -5833.694} C_VEL
LIN {X 0,Y 504.811,Z 467.786,A -85,B 0,C 180,E1 -5834.352,E2 -5834.352} C_VEL
LIN {X 0,Y 504.294,Z 481.302,A -85,B 0,C 180,E1 -5835.163,E2 -5835.163} C_VEL
LIN {X 0,Y 503.896,Z 493.5,A -85,B 0,C 180,E1 -5836.079,E2 -5836.079} C_VEL
LIN {X 0,Y 503.433,Z 504.654,A -85,B 0,C 180,E1 -5837.094,E2 -5837.094} C_VEL
LIN {X 0,Y 503.087,Z 515.738,A -85,B 0,C 180,E1 -5838.318,E2 -5838.318} C_VEL
LIN {X 0,Y 502.753,Z 524.845,A -85,B 0,C 180,E1 -5839.53,E2 -5839.53} C_VEL
LIN {X 0,Y 502.507,Z 533.616,A -85,B 0,C 180,E1 -5840.948,E2 -5840.948} C_VEL
LIN {X 0,Y 502.331,Z 540.694,A -85,B 0,C 180,E1 -5842.363,E2 -5842.363} C_VEL
LIN {X 0,Y 502.281,Z 545.592,A -85,B 0,C 180,E1 -5843.574,E2 -5843.574} C_VEL
LIN {X 0,Y 502.21,Z 549.548,A -85,B 0,C 180,E1 -5844.782,E2 -5844.782} C_VEL
LIN {X 0,Y 502.199,Z 552.6,A -85,B 0,C 180,E1 -5845.988,E2 -5845.988} C_VEL
LIN {X 0,Y 502.148,Z 555.379,A -85,B 0,C 180,E1 -5847.594,E2 -5847.594} C_VEL
LIN {X 0,Y 502.052,Z 556.737,A -85,B 0,C 180,E1 -5849.199,E2 -5849.199} C_VEL
LIN {X 0,Y 502.08,Z 556.717,A -85,B 0,C 180,E1 -5850.803,E2 -5850.803} C_VEL
LIN {X 0,Y 502.155,Z 555.305,A -85,B 0,C 180,E1 -5852.407,E2 -5852.407} C_VEL
LIN {X 0,Y 502.219,Z 552.463,A -85,B 0,C 180,E1 -5854.013,E2 -5854.013} C_VEL
LIN {X 0,Y 502.272,Z 548.108,A -85,B 0,C 180,E1 -5855.622,E2 -5855.622} C_VEL
LIN {X 0,Y 502.3,Z 543.95,A -85,B 0,C 180,E1 -5856.791,E2 -5856.791} C_VEL
LIN {X 0,Y 502.461,Z 537.448,A -85,B 0,C 180,E1 -5858.243,E2 -5858.243} C_VEL
LIN {X 0,Y 502.601,Z 529.51,A -85,B 0,C 180,E1 -5859.661,E2 -5859.661} C_VEL
LIN {X 0,Y 502.859,Z 521.249,A -85,B 0,C 180,E1 -5860.876,E2 -5860.876} C_VEL
LIN {X 0,Y 503.168,Z 511.102,A -85,B 0,C 180,E1 -5862.116,E2 -5862.116} C_VEL
LIN {X 0,Y 503.556,Z 499.166,A -85,B 0,C 180,E1 -5863.315,E2 -5863.315} C_VEL
LIN {X 0,Y 503.971,Z 486.795,A -85,B 0,C 180,E1 -5864.332,E2 -5864.332} C_VEL
LIN {X 0,Y 504.435,Z 474.712,A -85,B 0,C 180,E1 -5865.144,E2 -5865.144} C_VEL
LIN {X 0,Y 504.881,Z 461.612,A -85,B 0,C 180,E1 -5865.854,E2 -5865.854} C_VEL
LIN {X 0,Y 505.277,Z 447.29,A -85,B 0,C 180,E1 -5866.453,E2 -5866.453} C_VEL
LIN {X 0,Y 505.348,Z 437.253,A -85,B 0,C 180,E1 -5866.773,E2 -5866.773} C_VEL
LIN {X 0,Y 503.593,Z 425.976,A -85,B 0,C 180,E1 -5867.098,E2 -5867.098} C_VEL
LIN {X 0,Y 502.813,Z 418.204,A -85,B 0,C 180,E1 -5867.279,E2 -5867.279} C_VEL
LIN {X 0,Y 502.828,Z 416.685,A -85,B 0,C 180,E1 -5867.489,E2 -5867.489} C_VEL
LIN {X 0,Y 502.989,Z 401.769,A -85,B 0,C 180,E1 -5870.446,E2 -5870.446} C_VEL
LIN {X 0,Y 503.115,Z 385.555,A -85,B 0,C 180,E1 -5873.679,E2 -5873.679} C_VEL
LIN {X 0,Y 503.174,Z 370.982,A -85,B 0,C 180,E1 -5876.631,E2 -5876.631} C_VEL
LIN {X 0,Y 503.256,Z 358.278,A -85,B 0,C 180,E1 -5879.261,E2 -5879.261} C_VEL
LIN {X 0,Y 503.267,Z 344.182,A -85,B 0,C 180,E1 -5882.287,E2 -5882.287} C_VEL
LIN {X 0,Y 503.681,Z 328.014,A -85,B 0,C 180,E1 -5885.973,E2 -5885.973} C_VEL
LIN {X 0,Y 504.222,Z 318.822,A -85,B 0,C 180,E1 -5888.242,E2 -5888.242} C_VEL
LIN {X 0,Y 503.353,Z 313.198,A -85,B 0,C 180,E1 -5889.832,E2 -5889.832} C_VEL
LIN {X 0,Y 502.808,Z 310.555,A -85,B 0,C 180,E1 -5890.671,E2 -5890.671} C_VEL
LIN {X 0,Y 502.786,Z 310.484,A -85,B 0,C 180,E1 -5893.376,E2 -5893.376} C_VEL
LIN {X 0,Y 502.794,Z 310.484,A -85,B 0,C 180,E1 -5895.662,E2 -5895.662} C_VEL
LIN {X 0,Y 502.83,Z 310.476,A -85,B 0,C 180,E1 -5899.004,E2 -5899.004} C_VEL
LIN {X 0,Y 502.798,Z 310.479,A -85,B 0,C 180,E1 -5902.047,E2 -5902.047} C_VEL
LIN {X 0,Y 502.813,Z 310.477,A -85,B 0,C 180,E1 -5905.035,E2 -5905.035} C_VEL
LIN {X 0,Y 502.788,Z 310.48,A -85,B 0,C 180,E1 -5907.916,E2 -5907.916} C_VEL
LIN {X 0,Y 502.828,Z 310.473,A -85,B 0,C 180,E1 -5910.713,E2 -5910.713} C_VEL
LIN {X 0,Y 502.866,Z 310.475,A -85,B 0,C 180,E1 -5913.439,E2 -5913.439} C_VEL
LIN {X 0,Y 502.795,Z 310.478,A -85,B 0,C 180,E1 -5916.087,E2 -5916.087} C_VEL
LIN {X 0,Y 502.787,Z 310.482,A -85,B 0,C 180,E1 -5918.689,E2 -5918.689} C_VEL
LIN {X 0,Y 502.834,Z 310.479,A -85,B 0,C 180,E1 -5921.249,E2 -5921.249} C_VEL
LIN {X 0,Y 502.881,Z 310.606,A -85,B 0,C 180,E1 -5922.462,E2 -5922.462} C_VEL
LIN {X 0,Y 503.165,Z 311.79,A -85,B 0,C 180,E1 -5922.616,E2 -5922.616} C_VEL
LIN {X 0,Y 505.669,Z 320.008,A -85,B 0,C 180,E1 -5923.082,E2 -5923.082} C_VEL
LIN {X 0,Y 505.296,Z 332.589,A -85,B 0,C 180,E1 -5923.75,E2 -5923.75} C_VEL
LIN {X 0,Y 504.946,Z 344.747,A -85,B 0,C 180,E1 -5924.565,E2 -5924.565} C_VEL
LIN {X 0,Y 504.462,Z 355.864,A -85,B 0,C 180,E1 -5925.477,E2 -5925.477} C_VEL
LIN {X 0,Y 504.077,Z 366.075,A -85,B 0,C 180,E1 -5926.495,E2 -5926.495} C_VEL
LIN {X 0,Y 503.656,Z 375.54,A -85,B 0,C 180,E1 -5927.629,E2 -5927.629} C_VEL
LIN {X 0,Y 503.336,Z 384.484,A -85,B 0,C 180,E1 -5928.931,E2 -5928.931} C_VEL
LIN {X 0,Y 502.982,Z 392.368,A -85,B 0,C 180,E1 -5930.348,E2 -5930.348} C_VEL
LIN {X 0,Y 502.798,Z 397.864,A -85,B 0,C 180,E1 -5931.561,E2 -5931.561} C_VEL
LIN {X 0,Y 502.592,Z 403.503,A -85,B 0,C 180,E1 -5933.136,E2 -5933.136} C_VEL
LIN {X 0,Y 502.501,Z 406.893,A -85,B 0,C 180,E1 -5934.382,E2 -5934.382} C_VEL
LIN {X 0,Y 502.388,Z 410.009,A -85,B 0,C 180,E1 -5935.989,E2 -5935.989} C_VEL
LIN {X 0,Y 502.284,Z 411.768,A -85,B 0,C 180,E1 -5937.594,E2 -5937.594} C_VEL
LIN {X 0,Y 502.233,Z 412.216,A -85,B 0,C 180,E1 -5939.198,E2 -5939.198} C_VEL
LIN {X 0,Y 502.236,Z 411.372,A -85,B 0,C 180,E1 -5940.802,E2 -5940.802} C_VEL
LIN {X 0,Y 502.287,Z 409.216,A -85,B 0,C 180,E1 -5942.406,E2 -5942.406} C_VEL
LIN {X 0,Y 502.446,Z 405.694,A -85,B 0,C 180,E1 -5944.011,E2 -5944.011} C_VEL
LIN {X 0,Y 502.524,Z 400.719,A -85,B 0,C 180,E1 -5945.618,E2 -5945.618} C_VEL
LIN {X 0,Y 502.736,Z 395.116,A -85,B 0,C 180,E1 -5946.998,E2 -5946.998} C_VEL
LIN {X 0,Y 503,Z 387.835,A -85,B 0,C 180,E1 -5948.436,E2 -5948.436} C_VEL
LIN {X 0,Y 503.308,Z 378.961,A -85,B 0,C 180,E1 -5949.849,E2 -5949.849} C_VEL
LIN {X 0,Y 503.684,Z 369.62,A -85,B 0,C 180,E1 -5951.061,E2 -5951.061} C_VEL
LIN {X 0,Y 504.186,Z 358.217,A -85,B 0,C 180,E1 -5952.273,E2 -5952.273} C_VEL
LIN {X 0,Y 504.652,Z 346.561,A -85,B 0,C 180,E1 -5953.285,E2 -5953.285} C_VEL
LIN {X 0,Y 505.032,Z 335.169,A -85,B 0,C 180,E1 -5954.095,E2 -5954.095} C_VEL
LIN {X 0,Y 505.453,Z 321.438,A -85,B 0,C 180,E1 -5954.877,E2 -5954.877} C_VEL
LIN {X 0,Y 505.488,Z 319.479,A -85,B 0,C 180,E1 -5954.972,E2 -5954.972} C_VEL
LIN {X 0,Y 503.065,Z 311.522,A -85,B 0,C 180,E1 -5955.429,E2 -5955.429} C_VEL
LIN {X 0,Y 502.825,Z 310.521,A -85,B 0,C 180,E1 -5955.611,E2 -5955.611} C_VEL
LIN {X 0,Y 502.835,Z 310.478,A -85,B 0,C 180,E1 -5958.752,E2 -5958.752} C_VEL
LIN {X 0,Y 502.788,Z 310.48,A -85,B 0,C 180,E1 -5961.311,E2 -5961.311} C_VEL
LIN {X 0,Y 502.79,Z 310.477,A -85,B 0,C 180,E1 -5963.914,E2 -5963.914} C_VEL
LIN {X 0,Y 502.869,Z 310.472,A -85,B 0,C 180,E1 -5966.566,E2 -5966.566} C_VEL
LIN {X 0,Y 502.829,Z 310.472,A -85,B 0,C 180,E1 -5969.288,E2 -5969.288} C_VEL
LIN {X 0,Y 502.788,Z 310.477,A -85,B 0,C 180,E1 -5972.085,E2 -5972.085} C_VEL
LIN {X 0,Y 502.813,Z 310.476,A -85,B 0,C 180,E1 -5974.965,E2 -5974.965} C_VEL
LIN {X 0,Y 502.799,Z 310.476,A -85,B 0,C 180,E1 -5977.954,E2 -5977.954} C_VEL
LIN {X 0,Y 502.825,Z 310.472,A -85,B 0,C 180,E1 -5981.066,E2 -5981.066} C_VEL
LIN {X 0,Y 502.807,Z 310.481,A -85,B 0,C 180,E1 -5984.532,E2 -5984.532} C_VEL
LIN {X 0,Y 502.836,Z 310.472,A -85,B 0,C 180,E1 -5987.864,E2 -5987.864} C_VEL
LIN {X 0,Y 502.807,Z 310.474,A -85,B 0,C 180,E1 -5991.024,E2 -5991.024} C_VEL
LIN {X 0,Y 502.786,Z 310.479,A -85,B 0,C 180,E1 -5992.247,E2 -5992.247} C_VEL
LIN {X 0,Y 502.11,Z 310.563,A -85,B 0,C 180,E1 -5992.916,E2 -5992.916} C_VEL
LIN {X 0,Y 499.278,Z 310.917,A -85,B 0,C 180,E1 -5994.002,E2 -5994.002} C_VEL
LIN {X 0,Y 496.886,Z 311.212,A -85,B 0,C 180,E1 -5994.878,E2 -5994.878} C_VEL
LIN {X 0,Y 495.851,Z 311.34,A -85,B 0,C 180,E1 -5995.553,E2 -5995.553} C_VEL
LIN {X 0,Y 495.762,Z 311.351,A -85,B 0,C 180,E1 -5995.782,E2 -5995.782} C_VEL
LIN {X 0,Y 495.762,Z 311.357,A -85,B 0,C 180,E1 -5998.364,E2 -5998.364} C_VEL
LIN {X 0,Y 495.794,Z 311.348,A -85,B 0,C 180,E1 -6001.507,E2 -6001.507} C_VEL
LIN {X 0,Y 495.787,Z 311.353,A -85,B 0,C 180,E1 -6003.931,E2 -6003.931} C_VEL
LIN {X 0,Y 495.765,Z 311.35,A -85,B 0,C 180,E1 -6007.139,E2 -6007.139} C_VEL
LIN {X 0,Y 495.779,Z 311.357,A -85,B 0,C 180,E1 -6010.109,E2 -6010.109} C_VEL
LIN {X 0,Y 495.793,Z 311.348,A -85,B 0,C 180,E1 -6012.681,E2 -6012.681} C_VEL
LIN {X 0,Y 495.797,Z 311.347,A -85,B 0,C 180,E1 -6015.217,E2 -6015.217} C_VEL
LIN {X 0,Y 495.858,Z 311.34,A -85,B 0,C 180,E1 -6018.554,E2 -6018.554} C_VEL
LIN {X 0,Y 495.878,Z 311.345,A -85,B 0,C 180,E1 -6021.851,E2 -6021.851} C_VEL
LIN {X 0,Y 495.895,Z 311.337,A -85,B 0,C 180,E1 -6024.306,E2 -6024.306} C_VEL
LIN {X 0,Y 495.999,Z 311.327,A -85,B 0,C 180,E1 -6027.563,E2 -6027.563} C_VEL
LIN {X 0,Y 495.989,Z 311.323,A -85,B 0,C 180,E1 -6030.811,E2 -6030.811} C_VEL
LIN {X 0,Y 495.998,Z 311.322,A -85,B 0,C 180,E1 -6032.436,E2 -6032.436} C_VEL
LIN {X 0,Y 495.9,Z 311.342,A -85,B 0,C 180,E1 -6035.693,E2 -6035.693} C_VEL
LIN {X 0,Y 495.878,Z 311.338,A -85,B 0,C 180,E1 -6038.147,E2 -6038.147} C_VEL
LIN {X 0,Y 495.856,Z 311.346,A -85,B 0,C 180,E1 -6041.444,E2 -6041.444} C_VEL
LIN {X 0,Y 495.794,Z 311.347,A -85,B 0,C 180,E1 -6044.782,E2 -6044.782} C_VEL
LIN {X 0,Y 495.79,Z 311.354,A -85,B 0,C 180,E1 -6047.318,E2 -6047.318} C_VEL
LIN {X 0,Y 495.781,Z 311.351,A -85,B 0,C 180,E1 -6049.889,E2 -6049.889} C_VEL
LIN {X 0,Y 495.768,Z 311.352,A -85,B 0,C 180,E1 -6052.861,E2 -6052.861} C_VEL
LIN {X 0,Y 495.792,Z 311.348,A -85,B 0,C 180,E1 -6056.067,E2 -6056.067} C_VEL
LIN {X 0,Y 495.772,Z 311.352,A -85,B 0,C 180,E1 -6058.814,E2 -6058.814} C_VEL
LIN {X 0,Y 495.759,Z 311.354,A -85,B 0,C 180,E1 -6061.725,E2 -6061.725} C_VEL
LIN {X 0,Y 495.771,Z 311.352,A -85,B 0,C 180,E1 -6064.693,E2 -6064.693} C_VEL
LIN {X 0,Y 495.728,Z 311.358,A -85,B 0,C 180,E1 -6067.561,E2 -6067.561} C_VEL
LIN {X 0,Y 495.765,Z 311.353,A -85,B 0,C 180,E1 -6070.699,E2 -6070.699} C_VEL
LIN {X 0,Y 495.732,Z 311.356,A -85,B 0,C 180,E1 -6073.694,E2 -6073.694} C_VEL
LIN {X 0,Y 495.731,Z 311.355,A -85,B 0,C 180,E1 -6076.304,E2 -6076.304} C_VEL
LIN {X 0,Y 495.763,Z 311.355,A -85,B 0,C 180,E1 -6079.299,E2 -6079.299} C_VEL
LIN {X 0,Y 495.727,Z 311.357,A -85,B 0,C 180,E1 -6082.438,E2 -6082.438} C_VEL
LIN {X 0,Y 495.78,Z 311.35,A -85,B 0,C 180,E1 -6085.457,E2 -6085.457} C_VEL
LIN {X 0,Y 495.754,Z 311.354,A -85,B 0,C 180,E1 -6088.363,E2 -6088.363} C_VEL
LIN {X 0,Y 495.785,Z 311.349,A -85,B 0,C 180,E1 -6091.505,E2 -6091.505} C_VEL
LIN {X 0,Y 495.793,Z 311.347,A -85,B 0,C 180,E1 -6093.932,E2 -6093.932} C_VEL
LIN {X 0,Y 495.759,Z 311.354,A -85,B 0,C 180,E1 -6097.137,E2 -6097.137} C_VEL
LIN {X 0,Y 495.771,Z 311.351,A -85,B 0,C 180,E1 -6100.109,E2 -6100.109} C_VEL
LIN {X 0,Y 495.782,Z 311.357,A -85,B 0,C 180,E1 -6102.681,E2 -6102.681} C_VEL
LIN {X 0,Y 495.783,Z 311.349,A -85,B 0,C 180,E1 -6105.217,E2 -6105.217} C_VEL
LIN {X 0,Y 495.844,Z 311.35,A -85,B 0,C 180,E1 -6108.554,E2 -6108.554} C_VEL
LIN {X 0,Y 495.866,Z 311.339,A -85,B 0,C 180,E1 -6111.852,E2 -6111.852} C_VEL
LIN {X 0,Y 495.89,Z 311.341,A -85,B 0,C 180,E1 -6114.306,E2 -6114.306} C_VEL
LIN {X 0,Y 495.987,Z 311.323,A -85,B 0,C 180,E1 -6117.563,E2 -6117.563} C_VEL
LIN {X 0,Y 495.99,Z 311.326,A -85,B 0,C 180,E1 -6120,E2 -6120} C_VEL
LIN {X 0,Y 495.987,Z 311.33,A -85,B 0,C 180,E1 -6122.436,E2 -6122.436} C_VEL
LIN {X 0,Y 495.889,Z 311.336,A -85,B 0,C 180,E1 -6125.693,E2 -6125.693} C_VEL
LIN {X 0,Y 495.865,Z 311.345,A -85,B 0,C 180,E1 -6128.148,E2 -6128.148} C_VEL
LIN {X 0,Y 495.866,Z 311.338,A -85,B 0,C 180,E1 -6131.445,E2 -6131.445} C_VEL
LIN {X 0,Y 495.782,Z 311.349,A -85,B 0,C 180,E1 -6134.783,E2 -6134.783} C_VEL
LIN {X 0,Y 495.78,Z 311.349,A -85,B 0,C 180,E1 -6137.319,E2 -6137.319} C_VEL
LIN {X 0,Y 495.764,Z 311.356,A -85,B 0,C 180,E1 -6139.891,E2 -6139.891} C_VEL
LIN {X 0,Y 495.757,Z 311.352,A -85,B 0,C 180,E1 -6142.863,E2 -6142.863} C_VEL
LIN {X 0,Y 495.784,Z 311.356,A -85,B 0,C 180,E1 -6146.068,E2 -6146.068} C_VEL
LIN {X 0,Y 495.773,Z 311.35,A -85,B 0,C 180,E1 -6148.815,E2 -6148.815} C_VEL
LIN {X 0,Y 495.752,Z 311.358,A -85,B 0,C 180,E1 -6151.727,E2 -6151.727} C_VEL
LIN {X 0,Y 495.77,Z 311.35,A -85,B 0,C 180,E1 -6154.696,E2 -6154.696} C_VEL
LIN {X 0,Y 495.727,Z 311.362,A -85,B 0,C 180,E1 -6157.562,E2 -6157.562} C_VEL
LIN {X 0,Y 495.787,Z 311.355,A -85,B 0,C 180,E1 -6160.053,E2 -6160.053} C_VEL
LIN {X 0,Y 495.72,Z 311.361,A -85,B 0,C 180,E1 -6162.884,E2 -6162.884} C_VEL
LIN {X 0,Y 495.732,Z 311.362,A -85,B 0,C 180,E1 -6166,E2 -6166} C_VEL
LIN {X 0,Y 495.774,Z 311.556,A -85,B 0,C 180,E1 -6166.747,E2 -6166.747} C_VEL
LIN {X 0,Y 497.474,Z 319.397,A -85,B 0,C 180,E1 -6169.01,E2 -6169.01} C_VEL
LIN {X 0,Y 498.659,Z 325.931,A -85,B 0,C 180,E1 -6170.819,E2 -6170.819} C_VEL
LIN {X 0,Y 498.433,Z 333.215,A -85,B 0,C 180,E1 -6172.678,E2 -6172.678} C_VEL
LIN {X 0,Y 497.853,Z 345.137,A -85,B 0,C 180,E1 -6175.622,E2 -6175.622} C_VEL
LIN {X 0,Y 497.309,Z 359.012,A -85,B 0,C 180,E1 -6178.949,E2 -6178.949} C_VEL
LIN {X 0,Y 496.933,Z 370.898,A -85,B 0,C 180,E1 -6181.721,E2 -6181.721} C_VEL
LIN {X 0,Y 496.607,Z 382.79,A -85,B 0,C 180,E1 -6184.43,E2 -6184.43} C_VEL
LIN {X 0,Y 496.311,Z 395.431,A -85,B 0,C 180,E1 -6187.251,E2 -6187.251} C_VEL
LIN {X 0,Y 495.96,Z 410.538,A -85,B 0,C 180,E1 -6190.55,E2 -6190.55} C_VEL
LIN {X 0,Y 495.825,Z 419.385,A -85,B 0,C 180,E1 -6192.418,E2 -6192.418} C_VEL
LIN {X 0,Y 496.246,Z 422.82,A -85,B 0,C 180,E1 -6192.536,E2 -6192.536} C_VEL
LIN {X 0,Y 498.168,Z 435.771,A -85,B 0,C 180,E1 -6192.884,E2 -6192.884} C_VEL
LIN {X 0,Y 498.817,Z 439.847,A -85,B 0,C 180,E1 -6193.023,E2 -6193.023} C_VEL
LIN {X 0,Y 498.339,Z 454.243,A -85,B 0,C 180,E1 -6193.535,E2 -6193.535} C_VEL
LIN {X 0,Y 497.901,Z 466.8,A -85,B 0,C 180,E1 -6194.136,E2 -6194.136} C_VEL
LIN {X 0,Y 497.372,Z 480.233,A -85,B 0,C 180,E1 -6194.952,E2 -6194.952} C_VEL
LIN {X 0,Y 496.879,Z 492.442,A -85,B 0,C 180,E1 -6195.879,E2 -6195.879} C_VEL
LIN {X 0,Y 496.425,Z 503.616,A -85,B 0,C 180,E1 -6196.909,E2 -6196.909} C_VEL
LIN {X 0,Y 496.056,Z 513.272,A -85,B 0,C 180,E1 -6197.972,E2 -6197.972} C_VEL
LIN {X 0,Y 495.77,Z 522.444,A -85,B 0,C 180,E1 -6199.175,E2 -6199.175} C_VEL
LIN {X 0,Y 495.488,Z 531.47,A -85,B 0,C 180,E1 -6200.613,E2 -6200.613} C_VEL
LIN {X 0,Y 495.334,Z 537.842,A -85,B 0,C 180,E1 -6201.844,E2 -6201.844} C_VEL
LIN {X 0,Y 495.25,Z 544.615,A -85,B 0,C 180,E1 -6203.482,E2 -6203.482} C_VEL
LIN {X 0,Y 495.146,Z 549.674,A -85,B 0,C 180,E1 -6205.115,E2 -6205.115} C_VEL
LIN {X 0,Y 495.129,Z 553.188,A -85,B 0,C 180,E1 -6206.746,E2 -6206.746} C_VEL
LIN {X 0,Y 495.048,Z 555.241,A -85,B 0,C 180,E1 -6208.374,E2 -6208.374} C_VEL
LIN {X 0,Y 495.064,Z 555.904,A -85,B 0,C 180,E1 -6210.001,E2 -6210.001} C_VEL
LIN {X 0,Y 495.058,Z 555.159,A -85,B 0,C 180,E1 -6211.628,E2 -6211.628} C_VEL
LIN {X 0,Y 495.148,Z 553.014,A -85,B 0,C 180,E1 -6213.255,E2 -6213.255} C_VEL
LIN {X 0,Y 495.153,Z 550.443,A -85,B 0,C 180,E1 -6214.478,E2 -6214.478} C_VEL
LIN {X 0,Y 495.231,Z 546.024,A -85,B 0,C 180,E1 -6216.003,E2 -6216.003} C_VEL
LIN {X 0,Y 495.273,Z 540.948,A -85,B 0,C 180,E1 -6217.338,E2 -6217.338} C_VEL
LIN {X 0,Y 495.407,Z 534.125,A -85,B 0,C 180,E1 -6218.773,E2 -6218.773} C_VEL
LIN {X 0,Y 495.606,Z 525.65,A -85,B 0,C 180,E1 -6220.211,E2 -6220.211} C_VEL
LIN {X 0,Y 495.947,Z 516.814,A -85,B 0,C 180,E1 -6221.444,E2 -6221.444} C_VEL
LIN {X 0,Y 496.261,Z 506.148,A -85,B 0,C 180,E1 -6222.681,E2 -6222.681} C_VEL
LIN {X 0,Y 496.698,Z 494.244,A -85,B 0,C 180,E1 -6223.815,E2 -6223.815} C_VEL
LIN {X 0,Y 497.121,Z 482.436,A -85,B 0,C 180,E1 -6224.743,E2 -6224.743} C_VEL
LIN {X 0,Y 497.602,Z 469.606,A -85,B 0,C 180,E1 -6225.567,E2 -6225.567} C_VEL
LIN {X 0,Y 498.047,Z 456.6,A -85,B 0,C 180,E1 -6226.234,E2 -6226.234} C_VEL
LIN {X 0,Y 498.476,Z 442.194,A -85,B 0,C 180,E1 -6226.8,E2 -6226.8} C_VEL
LIN {X 0,Y 498.343,Z 437.767,A -85,B 0,C 180,E1 -6226.946,E2 -6226.946} C_VEL
LIN {X 0,Y 496.749,Z 426.824,A -85,B 0,C 180,E1 -6227.285,E2 -6227.285} C_VEL
LIN {X 0,Y 495.759,Z 416.712,A -85,B 0,C 180,E1 -6227.533,E2 -6227.533} C_VEL
LIN {X 0,Y 495.759,Z 415.282,A -85,B 0,C 180,E1 -6227.746,E2 -6227.746} C_VEL
LIN {X 0,Y 495.912,Z 401.56,A -85,B 0,C 180,E1 -6230.509,E2 -6230.509} C_VEL
LIN {X 0,Y 496.04,Z 385.263,A -85,B 0,C 180,E1 -6233.816,E2 -6233.816} C_VEL
LIN {X 0,Y 496.106,Z 372.585,A -85,B 0,C 180,E1 -6236.43,E2 -6236.43} C_VEL
LIN {X 0,Y 496.192,Z 359.211,A -85,B 0,C 180,E1 -6239.253,E2 -6239.253} C_VEL
LIN {X 0,Y 496.243,Z 347.455,A -85,B 0,C 180,E1 -6241.816,E2 -6241.816} C_VEL
LIN {X 0,Y 496.569,Z 331.606,A -85,B 0,C 180,E1 -6245.471,E2 -6245.471} C_VEL
LIN {X 0,Y 497.251,Z 321.412,A -85,B 0,C 180,E1 -6248.008,E2 -6248.008} C_VEL
LIN {X 0,Y 496.925,Z 317.126,A -85,B 0,C 180,E1 -6249.196,E2 -6249.196} C_VEL
LIN {X 0,Y 495.793,Z 311.426,A -85,B 0,C 180,E1 -6250.994,E2 -6250.994} C_VEL
LIN {X 0,Y 495.74,Z 311.362,A -85,B 0,C 180,E1 -6254.001,E2 -6254.001} C_VEL
LIN {X 0,Y 495.729,Z 311.362,A -85,B 0,C 180,E1 -6257.117,E2 -6257.117} C_VEL
LIN {X 0,Y 495.793,Z 311.354,A -85,B 0,C 180,E1 -6259.949,E2 -6259.949} C_VEL
LIN {X 0,Y 495.735,Z 311.358,A -85,B 0,C 180,E1 -6262.553,E2 -6262.553} C_VEL
LIN {X 0,Y 495.789,Z 311.355,A -85,B 0,C 180,E1 -6265.458,E2 -6265.458} C_VEL
LIN {X 0,Y 495.759,Z 311.353,A -85,B 0,C 180,E1 -6268.364,E2 -6268.364} C_VEL
LIN {X 0,Y 495.791,Z 311.354,A -85,B 0,C 180,E1 -6271.507,E2 -6271.507} C_VEL
LIN {X 0,Y 495.794,Z 311.351,A -85,B 0,C 180,E1 -6273.932,E2 -6273.932} C_VEL
LIN {X 0,Y 495.762,Z 311.359,A -85,B 0,C 180,E1 -6277.14,E2 -6277.14} C_VEL
LIN {X 0,Y 495.781,Z 311.355,A -85,B 0,C 180,E1 -6280.11,E2 -6280.11} C_VEL
LIN {X 0,Y 495.863,Z 311.565,A -85,B 0,C 180,E1 -6282.232,E2 -6282.232} C_VEL
LIN {X 0,Y 496.104,Z 312.584,A -85,B 0,C 180,E1 -6282.364,E2 -6282.364} C_VEL
LIN {X 0,Y 498.926,Z 321.676,A -85,B 0,C 180,E1 -6282.9,E2 -6282.9} C_VEL
LIN {X 0,Y 498.46,Z 334.905,A -85,B 0,C 180,E1 -6283.621,E2 -6283.621} C_VEL
LIN {X 0,Y 498.062,Z 346.854,A -85,B 0,C 180,E1 -6284.449,E2 -6284.449} C_VEL
LIN {X 0,Y 497.584,Z 358.921,A -85,B 0,C 180,E1 -6285.481,E2 -6285.481} C_VEL
LIN {X 0,Y 497.142,Z 368.8,A -85,B 0,C 180,E1 -6286.511,E2 -6286.511} C_VEL
LIN {X 0,Y 496.675,Z 378.575,A -85,B 0,C 180,E1 -6287.746,E2 -6287.746} C_VEL
LIN {X 0,Y 496.384,Z 386.64,A -85,B 0,C 180,E1 -6288.981,E2 -6288.981} C_VEL
LIN {X 0,Y 496.049,Z 393.345,A -85,B 0,C 180,E1 -6290.211,E2 -6290.211} C_VEL
LIN {X 0,Y 495.843,Z 398.848,A -85,B 0,C 180,E1 -6291.441,E2 -6291.441} C_VEL
LIN {X 0,Y 495.618,Z 404.508,A -85,B 0,C 180,E1 -6293.036,E2 -6293.036} C_VEL
LIN {X 0,Y 495.509,Z 407.908,A -85,B 0,C 180,E1 -6294.302,E2 -6294.302} C_VEL
LIN {X 0,Y 495.373,Z 411.039,A -85,B 0,C 180,E1 -6295.932,E2 -6295.932} C_VEL
LIN {X 0,Y 495.264,Z 412.796,A -85,B 0,C 180,E1 -6297.56,E2 -6297.56} C_VEL
LIN {X 0,Y 495.217,Z 413.232,A -85,B 0,C 180,E1 -6299.187,E2 -6299.187} C_VEL
LIN {X 0,Y 495.22,Z 412.375,A -85,B 0,C 180,E1 -6300.813,E2 -6300.813} C_VEL
LIN {X 0,Y 495.264,Z 410.208,A -85,B 0,C 180,E1 -6302.44,E2 -6302.44} C_VEL
LIN {X 0,Y 495.431,Z 406.667,A -85,B 0,C 180,E1 -6304.068,E2 -6304.068} C_VEL
LIN {X 0,Y 495.527,Z 401.672,A -85,B 0,C 180,E1 -6305.698,E2 -6305.698} C_VEL
LIN {X 0,Y 495.761,Z 396.05,A -85,B 0,C 180,E1 -6307.097,E2 -6307.097} C_VEL
LIN {X 0,Y 496.045,Z 388.746,A -85,B 0,C 180,E1 -6308.556,E2 -6308.556} C_VEL
LIN {X 0,Y 496.371,Z 379.846,A -85,B 0,C 180,E1 -6309.988,E2 -6309.988} C_VEL
LIN {X 0,Y 496.772,Z 370.484,A -85,B 0,C 180,E1 -6311.217,E2 -6311.217} C_VEL
LIN {X 0,Y 497.309,Z 359.083,A -85,B 0,C 180,E1 -6312.443,E2 -6312.443} C_VEL
LIN {X 0,Y 497.809,Z 347.39,A -85,B 0,C 180,E1 -6313.471,E2 -6313.471} C_VEL
LIN {X 0,Y 498.21,Z 335.993,A -85,B 0,C 180,E1 -6314.292,E2 -6314.292} C_VEL
LIN {X 0,Y 498.618,Z 323.193,A -85,B 0,C 180,E1 -6315.036,E2 -6315.036} C_VEL
LIN {X 0,Y 498.351,Z 319.877,A -85,B 0,C 180,E1 -6315.214,E2 -6315.214} C_VEL
LIN {X 0,Y 495.889,Z 311.96,A -85,B 0,C 180,E1 -6315.701,E2 -6315.701} C_VEL
LIN {X 0,Y 495.788,Z 311.401,A -85,B 0,C 180,E1 -6315.836,E2 -6315.836} C_VEL
LIN {X 0,Y 495.789,Z 311.356,A -85,B 0,C 180,E1 -6319.029,E2 -6319.029} C_VEL
LIN {X 0,Y 495.747,Z 311.355,A -85,B 0,C 180,E1 -6321.629,E2 -6321.629} C_VEL
LIN {X 0,Y 495.783,Z 311.355,A -85,B 0,C 180,E1 -6324.873,E2 -6324.873} C_VEL
LIN {X 0,Y 495.818,Z 311.348,A -85,B 0,C 180,E1 -6326.974,E2 -6326.974} C_VEL
LIN {X 0,Y 495.77,Z 311.352,A -85,B 0,C 180,E1 -6330.147,E2 -6330.147} C_VEL
LIN {X 0,Y 495.798,Z 311.347,A -85,B 0,C 180,E1 -6333.245,E2 -6333.245} C_VEL
LIN {X 0,Y 495.732,Z 311.357,A -85,B 0,C 180,E1 -6336.09,E2 -6336.09} C_VEL
LIN {X 0,Y 495.769,Z 311.355,A -85,B 0,C 180,E1 -6338.768,E2 -6338.768} C_VEL
LIN {X 0,Y 495.761,Z 311.352,A -85,B 0,C 180,E1 -6341.781,E2 -6341.781} C_VEL
LIN {X 0,Y 495.755,Z 311.352,A -85,B 0,C 180,E1 -6345.139,E2 -6345.139} C_VEL
LIN {X 0,Y 495.783,Z 311.355,A -85,B 0,C 180,E1 -6348.221,E2 -6348.221} C_VEL
LIN {X 0,Y 495.755,Z 311.352,A -85,B 0,C 180,E1 -6351.408,E2 -6351.408} C_VEL
LIN {X 0,Y 495.754,Z 311.358,A -85,B 0,C 180,E1 -6354.462,E2 -6354.462} C_VEL
LIN {X 0,Y 495.762,Z 311.351,A -85,B 0,C 180,E1 -6355.782,E2 -6355.782} C_VEL
LIN {X 0,Y 495.075,Z 311.442,A -85,B 0,C 180,E1 -6356.46,E2 -6356.46} C_VEL
LIN {X 0,Y 492.197,Z 311.796,A -85,B 0,C 180,E1 -6357.562,E2 -6357.562} C_VEL
LIN {X 0,Y 489.786,Z 312.1,A -85,B 0,C 180,E1 -6358.449,E2 -6358.449} C_VEL
LIN {X 0,Y 488.771,Z 312.222,A -85,B 0,C 180,E1 -6359.135,E2 -6359.135} C_VEL
LIN {X 0,Y 488.699,Z 312.231,A -85,B 0,C 180,E1 -6359.367,E2 -6359.367} C_VEL
LIN {X 0,Y 488.753,Z 312.227,A -85,B 0,C 180,E1 -6362.603,E2 -6362.603} C_VEL
LIN {X 0,Y 488.722,Z 312.228,A -85,B 0,C 180,E1 -6365.352,E2 -6365.352} C_VEL
LIN {X 0,Y 488.705,Z 312.238,A -85,B 0,C 180,E1 -6368.043,E2 -6368.043} C_VEL
LIN {X 0,Y 488.75,Z 312.225,A -85,B 0,C 180,E1 -6370.686,E2 -6370.686} C_VEL
LIN {X 0,Y 488.737,Z 312.227,A -85,B 0,C 180,E1 -6373.285,E2 -6373.285} C_VEL
LIN {X 0,Y 488.745,Z 312.232,A -85,B 0,C 180,E1 -6375.85,E2 -6375.85} C_VEL
LIN {X 0,Y 488.812,Z 312.219,A -85,B 0,C 180,E1 -6378.387,E2 -6378.387} C_VEL
LIN {X 0,Y 488.822,Z 312.222,A -85,B 0,C 180,E1 -6381.733,E2 -6381.733} C_VEL
LIN {X 0,Y 488.853,Z 312.215,A -85,B 0,C 180,E1 -6384.224,E2 -6384.224} C_VEL
LIN {X 0,Y 488.967,Z 312.202,A -85,B 0,C 180,E1 -6387.528,E2 -6387.528} C_VEL
LIN {X 0,Y 488.94,Z 312.201,A -85,B 0,C 180,E1 -6390.823,E2 -6390.823} C_VEL
LIN {X 0,Y 488.966,Z 312.198,A -85,B 0,C 180,E1 -6392.471,E2 -6392.471} C_VEL
LIN {X 0,Y 488.859,Z 312.218,A -85,B 0,C 180,E1 -6395.775,E2 -6395.775} C_VEL
LIN {X 0,Y 488.822,Z 312.216,A -85,B 0,C 180,E1 -6398.265,E2 -6398.265} C_VEL
LIN {X 0,Y 488.81,Z 312.225,A -85,B 0,C 180,E1 -6401.611,E2 -6401.611} C_VEL
LIN {X 0,Y 488.765,Z 312.224,A -85,B 0,C 180,E1 -6404.999,E2 -6404.999} C_VEL
LIN {X 0,Y 488.758,Z 312.223,A -85,B 0,C 180,E1 -6408.441,E2 -6408.441} C_VEL
LIN {X 0,Y 488.709,Z 312.233,A -85,B 0,C 180,E1 -6411.07,E2 -6411.07} C_VEL
LIN {X 0,Y 488.695,Z 312.235,A -85,B 0,C 180,E1 -6413.744,E2 -6413.744} C_VEL
LIN {X 0,Y 488.793,Z 312.222,A -85,B 0,C 180,E1 -6416.943,E2 -6416.943} C_VEL
LIN {X 0,Y 488.71,Z 312.229,A -85,B 0,C 180,E1 -6420.362,E2 -6420.362} C_VEL
LIN {X 0,Y 488.735,Z 312.231,A -85,B 0,C 180,E1 -6423.483,E2 -6423.483} C_VEL
LIN {X 0,Y 488.681,Z 312.233,A -85,B 0,C 180,E1 -6426.354,E2 -6426.354} C_VEL
LIN {X 0,Y 488.7,Z 312.238,A -85,B 0,C 180,E1 -6429.253,E2 -6429.253} C_VEL
LIN {X 0,Y 488.721,Z 312.23,A -85,B 0,C 180,E1 -6431.601,E2 -6431.601} C_VEL
LIN {X 0,Y 488.709,Z 312.234,A -85,B 0,C 180,E1 -6434.8,E2 -6434.8} C_VEL
LIN {X 0,Y 488.692,Z 312.234,A -85,B 0,C 180,E1 -6437.474,E2 -6437.474} C_VEL
LIN {X 0,Y 488.729,Z 312.228,A -85,B 0,C 180,E1 -6439.676,E2 -6439.676} C_VEL
LIN {X 0,Y 488.678,Z 312.24,A -85,B 0,C 180,E1 -6442.841,E2 -6442.841} C_VEL
LIN {X 0,Y 488.73,Z 312.227,A -85,B 0,C 180,E1 -6445.887,E2 -6445.887} C_VEL
LIN {X 0,Y 488.713,Z 312.237,A -85,B 0,C 180,E1 -6448.821,E2 -6448.821} C_VEL
LIN {X 0,Y 488.741,Z 312.225,A -85,B 0,C 180,E1 -6451.671,E2 -6451.671} C_VEL
LIN {X 0,Y 488.745,Z 312.229,A -85,B 0,C 180,E1 -6454.444,E2 -6454.444} C_VEL
LIN {X 0,Y 488.721,Z 312.231,A -85,B 0,C 180,E1 -6457.153,E2 -6457.153} C_VEL
LIN {X 0,Y 488.722,Z 312.228,A -85,B 0,C 180,E1 -6459.81,E2 -6459.81} C_VEL
LIN {X 0,Y 488.729,Z 312.232,A -85,B 0,C 180,E1 -6462.423,E2 -6462.423} C_VEL
LIN {X 0,Y 488.755,Z 312.227,A -85,B 0,C 180,E1 -6464.999,E2 -6464.999} C_VEL
LIN {X 0,Y 488.798,Z 312.224,A -85,B 0,C 180,E1 -6468.387,E2 -6468.387} C_VEL
LIN {X 0,Y 488.81,Z 312.217,A -85,B 0,C 180,E1 -6471.733,E2 -6471.733} C_VEL
LIN {X 0,Y 488.849,Z 312.217,A -85,B 0,C 180,E1 -6474.224,E2 -6474.224} C_VEL
LIN {X 0,Y 488.955,Z 312.199,A -85,B 0,C 180,E1 -6477.528,E2 -6477.528} C_VEL
LIN {X 0,Y 488.969,Z 312.2,A -85,B 0,C 180,E1 -6480.823,E2 -6480.823} C_VEL
LIN {X 0,Y 488.954,Z 312.206,A -85,B 0,C 180,E1 -6482.471,E2 -6482.471} C_VEL
LIN {X 0,Y 488.848,Z 312.214,A -85,B 0,C 180,E1 -6485.776,E2 -6485.776} C_VEL
LIN {X 0,Y 488.81,Z 312.226,A -85,B 0,C 180,E1 -6488.266,E2 -6488.266} C_VEL
LIN {X 0,Y 488.824,Z 312.216,A -85,B 0,C 180,E1 -6491.612,E2 -6491.612} C_VEL
LIN {X 0,Y 488.754,Z 312.224,A -85,B 0,C 180,E1 -6495,E2 -6495} C_VEL
LIN {X 0,Y 488.747,Z 312.229,A -85,B 0,C 180,E1 -6498.442,E2 -6498.442} C_VEL
LIN {X 0,Y 488.699,Z 312.231,A -85,B 0,C 180,E1 -6501.071,E2 -6501.071} C_VEL
LIN {X 0,Y 488.686,Z 312.237,A -85,B 0,C 180,E1 -6503.746,E2 -6503.746} C_VEL
LIN {X 0,Y 488.784,Z 312.22,A -85,B 0,C 180,E1 -6506.944,E2 -6506.944} C_VEL
LIN {X 0,Y 488.727,Z 312.232,A -85,B 0,C 180,E1 -6510.219,E2 -6510.219} C_VEL
LIN {X 0,Y 488.729,Z 312.23,A -85,B 0,C 180,E1 -6513.485,E2 -6513.485} C_VEL
LIN {X 0,Y 488.683,Z 312.237,A -85,B 0,C 180,E1 -6516.356,E2 -6516.356} C_VEL
LIN {X 0,Y 488.742,Z 312.23,A -85,B 0,C 180,E1 -6519.25,E2 -6519.25} C_VEL
LIN {X 0,Y 488.685,Z 312.237,A -85,B 0,C 180,E1 -6522.526,E2 -6522.526} C_VEL
LIN {X 0,Y 488.706,Z 312.238,A -85,B 0,C 180,E1 -6525.199,E2 -6525.199} C_VEL
LIN {X 0,Y 488.737,Z 312.414,A -85,B 0,C 180,E1 -6526.413,E2 -6526.413} C_VEL
LIN {X 0,Y 490.637,Z 321.25,A -85,B 0,C 180,E1 -6529.001,E2 -6529.001} C_VEL
LIN {X 0,Y 491.665,Z 326.66,A -85,B 0,C 180,E1 -6530.524,E2 -6530.524} C_VEL
LIN {X 0,Y 491.668,Z 332.559,A -85,B 0,C 180,E1 -6532.075,E2 -6532.075} C_VEL
LIN {X 0,Y 490.899,Z 346.459,A -85,B 0,C 180,E1 -6535.564,E2 -6535.564} C_VEL
LIN {X 0,Y 490.311,Z 360.327,A -85,B 0,C 180,E1 -6538.936,E2 -6538.936} C_VEL
LIN {X 0,Y 489.905,Z 372.191,A -85,B 0,C 180,E1 -6541.745,E2 -6541.745} C_VEL
LIN {X 0,Y 489.524,Z 385.216,A -85,B 0,C 180,E1 -6544.753,E2 -6544.753} C_VEL
LIN {X 0,Y 489.276,Z 395.931,A -85,B 0,C 180,E1 -6547.181,E2 -6547.181} C_VEL
LIN {X 0,Y 488.91,Z 409.746,A -85,B 0,C 180,E1 -6550.258,E2 -6550.258} C_VEL
LIN {X 0,Y 488.744,Z 418.55,A -85,B 0,C 180,E1 -6552.156,E2 -6552.156} C_VEL
LIN {X 0,Y 489.071,Z 421.074,A -85,B 0,C 180,E1 -6552.262,E2 -6552.262} C_VEL
LIN {X 0,Y 491.118,Z 435.627,A -85,B 0,C 180,E1 -6552.66,E2 -6552.66} C_VEL
LIN {X 0,Y 491.907,Z 441.441,A -85,B 0,C 180,E1 -6552.863,E2 -6552.863} C_VEL
LIN {X 0,Y 491.405,Z 455.039,A -85,B 0,C 180,E1 -6553.38,E2 -6553.38} C_VEL
LIN {X 0,Y 490.927,Z 467.888,A -85,B 0,C 180,E1 -6554.028,E2 -6554.028} C_VEL
LIN {X 0,Y 490.371,Z 480.62,A -85,B 0,C 180,E1 -6554.838,E2 -6554.838} C_VEL
LIN {X 0,Y 489.845,Z 492.586,A -85,B 0,C 180,E1 -6555.778,E2 -6555.778} C_VEL
LIN {X 0,Y 489.413,Z 502.577,A -85,B 0,C 180,E1 -6556.718,E2 -6556.718} C_VEL
LIN {X 0,Y 488.969,Z 513.217,A -85,B 0,C 180,E1 -6557.917,E2 -6557.917} C_VEL
LIN {X 0,Y 488.68,Z 522.828,A -85,B 0,C 180,E1 -6559.225,E2 -6559.225} C_VEL
LIN {X 0,Y 488.388,Z 531.615,A -85,B 0,C 180,E1 -6560.684,E2 -6560.684} C_VEL
LIN {X 0,Y 488.201,Z 538.712,A -85,B 0,C 180,E1 -6562.14,E2 -6562.14} C_VEL
LIN {X 0,Y 488.176,Z 544.69,A -85,B 0,C 180,E1 -6563.688,E2 -6563.688} C_VEL
LIN {X 0,Y 488.098,Z 548.694,A -85,B 0,C 180,E1 -6565.045,E2 -6565.045} C_VEL
LIN {X 0,Y 488.082,Z 552.205,A -85,B 0,C 180,E1 -6566.699,E2 -6566.699} C_VEL
LIN {X 0,Y 488.014,Z 554.253,A -85,B 0,C 180,E1 -6568.35,E2 -6568.35} C_VEL
LIN {X 0,Y 488.054,Z 554.905,A -85,B 0,C 180,E1 -6570.001,E2 -6570.001} C_VEL
LIN {X 0,Y 488.029,Z 554.136,A -85,B 0,C 180,E1 -6571.651,E2 -6571.651} C_VEL
LIN {X 0,Y 488.11,Z 551.962,A -85,B 0,C 180,E1 -6573.302,E2 -6573.302} C_VEL
LIN {X 0,Y 488.136,Z 549.364,A -85,B 0,C 180,E1 -6574.543,E2 -6574.543} C_VEL
LIN {X 0,Y 488.166,Z 545.892,A -85,B 0,C 180,E1 -6575.785,E2 -6575.785} C_VEL
LIN {X 0,Y 488.199,Z 541.488,A -85,B 0,C 180,E1 -6577.029,E2 -6577.029} C_VEL
LIN {X 0,Y 488.322,Z 535.043,A -85,B 0,C 180,E1 -6578.484,E2 -6578.484} C_VEL
LIN {X 0,Y 488.481,Z 526.998,A -85,B 0,C 180,E1 -6579.943,E2 -6579.943} C_VEL
LIN {X 0,Y 488.752,Z 518.618,A -85,B 0,C 180,E1 -6581.194,E2 -6581.194} C_VEL
LIN {X 0,Y 489.084,Z 508.526,A -85,B 0,C 180,E1 -6582.448,E2 -6582.448} C_VEL
LIN {X 0,Y 489.491,Z 497.366,A -85,B 0,C 180,E1 -6583.599,E2 -6583.599} C_VEL
LIN {X 0,Y 489.994,Z 485.093,A -85,B 0,C 180,E1 -6584.644,E2 -6584.644} C_VEL
LIN {X 0,Y 490.537,Z 471.529,A -85,B 0,C 180,E1 -6585.584,E2 -6585.584} C_VEL
LIN {X 0,Y 491.049,Z 458.579,A -85,B 0,C 180,E1 -6586.299,E2 -6586.299} C_VEL
LIN {X 0,Y 491.514,Z 444.202,A -85,B 0,C 180,E1 -6586.912,E2 -6586.912} C_VEL
LIN {X 0,Y 491.398,Z 438.523,A -85,B 0,C 180,E1 -6587.117,E2 -6587.117} C_VEL
LIN {X 0,Y 489.909,Z 427.819,A -85,B 0,C 180,E1 -6587.466,E2 -6587.466} C_VEL
LIN {X 0,Y 488.668,Z 415.427,A -85,B 0,C 180,E1 -6587.789,E2 -6587.789} C_VEL
LIN {X 0,Y 488.698,Z 413.972,A -85,B 0,C 180,E1 -6587.997,E2 -6587.997} C_VEL
LIN {X 0,Y 488.811,Z 400.063,A -85,B 0,C 180,E1 -6590.844,E2 -6590.844} C_VEL
LIN {X 0,Y 488.97,Z 385.01,A -85,B 0,C 180,E1 -6593.957,E2 -6593.957} C_VEL
LIN {X 0,Y 489.04,Z 371.829,A -85,B 0,C 180,E1 -6596.729,E2 -6596.729} C_VEL
LIN {X 0,Y 489.146,Z 359.07,A -85,B 0,C 180,E1 -6599.479,E2 -6599.479} C_VEL
LIN {X 0,Y 489.237,Z 346.243,A -85,B 0,C 180,E1 -6602.352,E2 -6602.352} C_VEL
LIN {X 0,Y 489.663,Z 331.759,A -85,B 0,C 180,E1 -6605.794,E2 -6605.794} C_VEL
LIN {X 0,Y 490.332,Z 322.941,A -85,B 0,C 180,E1 -6608.049,E2 -6608.049} C_VEL
LIN {X 0,Y 490.043,Z 318.734,A -85,B 0,C 180,E1 -6609.245,E2 -6609.245} C_VEL
LIN {X 0,Y 488.749,Z 312.299,A -85,B 0,C 180,E1 -6611.346,E2 -6611.346} C_VEL
LIN {X 0,Y 488.706,Z 312.238,A -85,B 0,C 180,E1 -6614.025,E2 -6614.025} C_VEL
LIN {X 0,Y 488.713,Z 312.236,A -85,B 0,C 180,E1 -6617.174,E2 -6617.174} C_VEL
LIN {X 0,Y 488.737,Z 312.234,A -85,B 0,C 180,E1 -6619.677,E2 -6619.677} C_VEL
LIN {X 0,Y 488.684,Z 312.237,A -85,B 0,C 180,E1 -6622.278,E2 -6622.278} C_VEL
LIN {X 0,Y 488.732,Z 312.231,A -85,B 0,C 180,E1 -6625.052,E2 -6625.052} C_VEL
LIN {X 0,Y 488.707,Z 312.233,A -85,B 0,C 180,E1 -6628.046,E2 -6628.046} C_VEL
LIN {X 0,Y 488.727,Z 312.23,A -85,B 0,C 180,E1 -6630.73,E2 -6630.73} C_VEL
LIN {X 0,Y 488.761,Z 312.231,A -85,B 0,C 180,E1 -6633.528,E2 -6633.528} C_VEL
LIN {X 0,Y 488.697,Z 312.235,A -85,B 0,C 180,E1 -6636.255,E2 -6636.255} C_VEL
LIN {X 0,Y 488.75,Z 312.233,A -85,B 0,C 180,E1 -6639.176,E2 -6639.176} C_VEL
LIN {X 0,Y 488.807,Z 312.351,A -85,B 0,C 180,E1 -6641.944,E2 -6641.944} C_VEL
LIN {X 0,Y 489.116,Z 313.61,A -85,B 0,C 180,E1 -6642.116,E2 -6642.116} C_VEL
LIN {X 0,Y 492.119,Z 323.495,A -85,B 0,C 180,E1 -6642.709,E2 -6642.709} C_VEL
LIN {X 0,Y 491.676,Z 337.012,A -85,B 0,C 180,E1 -6643.472,E2 -6643.472} C_VEL
LIN {X 0,Y 491.238,Z 349.041,A -85,B 0,C 180,E1 -6644.334,E2 -6644.334} C_VEL
LIN {X 0,Y 490.763,Z 359.783,A -85,B 0,C 180,E1 -6645.275,E2 -6645.275} C_VEL
LIN {X 0,Y 490.304,Z 369.69,A -85,B 0,C 180,E1 -6646.319,E2 -6646.319} C_VEL
LIN {X 0,Y 489.791,Z 379.513,A -85,B 0,C 180,E1 -6647.571,E2 -6647.571} C_VEL
LIN {X 0,Y 489.475,Z 387.602,A -85,B 0,C 180,E1 -6648.823,E2 -6648.823} C_VEL
LIN {X 0,Y 489.122,Z 394.324,A -85,B 0,C 180,E1 -6650.071,E2 -6650.071} C_VEL
LIN {X 0,Y 488.891,Z 399.832,A -85,B 0,C 180,E1 -6651.319,E2 -6651.319} C_VEL
LIN {X 0,Y 488.646,Z 405.516,A -85,B 0,C 180,E1 -6652.934,E2 -6652.934} C_VEL
LIN {X 0,Y 488.518,Z 408.924,A -85,B 0,C 180,E1 -6654.22,E2 -6654.22} C_VEL
LIN {X 0,Y 488.359,Z 412.064,A -85,B 0,C 180,E1 -6655.874,E2 -6655.874} C_VEL
LIN {X 0,Y 488.244,Z 413.826,A -85,B 0,C 180,E1 -6657.525,E2 -6657.525} C_VEL
LIN {X 0,Y 488.2,Z 414.258,A -85,B 0,C 180,E1 -6659.175,E2 -6659.175} C_VEL
LIN {X 0,Y 488.203,Z 413.387,A -85,B 0,C 180,E1 -6660.825,E2 -6660.825} C_VEL
LIN {X 0,Y 488.241,Z 411.204,A -85,B 0,C 180,E1 -6662.475,E2 -6662.475} C_VEL
LIN {X 0,Y 488.417,Z 407.641,A -85,B 0,C 180,E1 -6664.126,E2 -6664.126} C_VEL
LIN {X 0,Y 488.531,Z 402.626,A -85,B 0,C 180,E1 -6665.78,E2 -6665.78} C_VEL
LIN {X 0,Y 488.787,Z 396.982,A -85,B 0,C 180,E1 -6667.199,E2 -6667.199} C_VEL
LIN {X 0,Y 489.092,Z 389.657,A -85,B 0,C 180,E1 -6668.678,E2 -6668.678} C_VEL
LIN {X 0,Y 489.414,Z 382.104,A -85,B 0,C 180,E1 -6669.923,E2 -6669.923} C_VEL
LIN {X 0,Y 489.784,Z 373.04,A -85,B 0,C 180,E1 -6671.17,E2 -6671.17} C_VEL
LIN {X 0,Y 490.295,Z 363.977,A -85,B 0,C 180,E1 -6672.206,E2 -6672.206} C_VEL
LIN {X 0,Y 490.77,Z 353.187,A -85,B 0,C 180,E1 -6673.246,E2 -6673.246} C_VEL
LIN {X 0,Y 491.239,Z 341.391,A -85,B 0,C 180,E1 -6674.182,E2 -6674.182} C_VEL
LIN {X 0,Y 491.721,Z 328.911,A -85,B 0,C 180,E1 -6674.983,E2 -6674.983} C_VEL
LIN {X 0,Y 491.729,Z 322.115,A -85,B 0,C 180,E1 -6675.354,E2 -6675.354} C_VEL
LIN {X 0,Y 488.857,Z 312.838,A -85,B 0,C 180,E1 -6675.932,E2 -6675.932} C_VEL
LIN {X 0,Y 488.753,Z 312.277,A -85,B 0,C 180,E1 -6676.07,E2 -6676.07} C_VEL
LIN {X 0,Y 488.748,Z 312.231,A -85,B 0,C 180,E1 -6679.313,E2 -6679.313} C_VEL
LIN {X 0,Y 488.703,Z 312.233,A -85,B 0,C 180,E1 -6681.957,E2 -6681.957} C_VEL
LIN {X 0,Y 488.749,Z 312.228,A -85,B 0,C 180,E1 -6685.053,E2 -6685.053} C_VEL
LIN {X 0,Y 488.751,Z 312.225,A -85,B 0,C 180,E1 -6687.397,E2 -6687.397} C_VEL
LIN {X 0,Y 488.714,Z 312.233,A -85,B 0,C 180,E1 -6690.363,E2 -6690.363} C_VEL
LIN {X 0,Y 488.74,Z 312.226,A -85,B 0,C 180,E1 -6693.484,E2 -6693.484} C_VEL
LIN {X 0,Y 488.693,Z 312.237,A -85,B 0,C 180,E1 -6696.355,E2 -6696.355} C_VEL
LIN {X 0,Y 488.706,Z 312.23,A -85,B 0,C 180,E1 -6699.254,E2 -6699.254} C_VEL
LIN {X 0,Y 488.712,Z 312.229,A -85,B 0,C 180,E1 -6701.6,E2 -6701.6} C_VEL
LIN {X 0,Y 488.718,Z 312.232,A -85,B 0,C 180,E1 -6704.801,E2 -6704.801} C_VEL
LIN {X 0,Y 488.701,Z 312.23,A -85,B 0,C 180,E1 -6707.475,E2 -6707.475} C_VEL
LIN {X 0,Y 488.739,Z 312.227,A -85,B 0,C 180,E1 -6709.677,E2 -6709.677} C_VEL
LIN {X 0,Y 488.685,Z 312.234,A -85,B 0,C 180,E1 -6712.841,E2 -6712.841} C_VEL
LIN {X 0,Y 488.736,Z 312.229,A -85,B 0,C 180,E1 -6715.887,E2 -6715.887} C_VEL
LIN {X 0,Y 488.698,Z 312.232,A -85,B 0,C 180,E1 -6718.82,E2 -6718.82} C_VEL
LIN {X 0,Y 488.699,Z 312.231,A -85,B 0,C 180,E1 -6719.367,E2 -6719.367} C_VEL
LIN {X 0,Y 488.067,Z 312.316,A -85,B 0,C 180,E1 -6720.055,E2 -6720.055} C_VEL
LIN {X 0,Y 485.253,Z 312.663,A -85,B 0,C 180,E1 -6721.171,E2 -6721.171} C_VEL
LIN {X 0,Y 482.859,Z 312.965,A -85,B 0,C 180,E1 -6722.072,E2 -6722.072} C_VEL
LIN {X 0,Y 481.833,Z 313.087,A -85,B 0,C 180,E1 -6722.767,E2 -6722.767} C_VEL
LIN {X 0,Y 481.751,Z 313.096,A -85,B 0,C 180,E1 -6723.002,E2 -6723.002} C_VEL
LIN {X 0,Y 481.668,Z 313.112,A -85,B 0,C 180,E1 -6725.886,E2 -6725.886} C_VEL
LIN {X 0,Y 481.709,Z 313.101,A -85,B 0,C 180,E1 -6729.027,E2 -6729.027} C_VEL
LIN {X 0,Y 481.714,Z 313.107,A -85,B 0,C 180,E1 -6732.158,E2 -6732.158} C_VEL
LIN {X 0,Y 481.749,Z 313.097,A -85,B 0,C 180,E1 -6734.775,E2 -6734.775} C_VEL
LIN {X 0,Y 481.757,Z 313.1,A -85,B 0,C 180,E1 -6738.215,E2 -6738.215} C_VEL
LIN {X 0,Y 481.768,Z 313.099,A -85,B 0,C 180,E1 -6741.611,E2 -6741.611} C_VEL
LIN {X 0,Y 481.814,Z 313.093,A -85,B 0,C 180,E1 -6744.139,E2 -6744.139} C_VEL
LIN {X 0,Y 481.933,Z 313.078,A -85,B 0,C 180,E1 -6747.492,E2 -6747.492} C_VEL
LIN {X 0,Y 481.892,Z 313.079,A -85,B 0,C 180,E1 -6750.835,E2 -6750.835} C_VEL
LIN {X 0,Y 481.933,Z 313.074,A -85,B 0,C 180,E1 -6752.507,E2 -6752.507} C_VEL
LIN {X 0,Y 481.82,Z 313.093,A -85,B 0,C 180,E1 -6755.86,E2 -6755.86} C_VEL
LIN {X 0,Y 481.767,Z 313.095,A -85,B 0,C 180,E1 -6758.387,E2 -6758.387} C_VEL
LIN {X 0,Y 481.755,Z 313.101,A -85,B 0,C 180,E1 -6761.784,E2 -6761.784} C_VEL
LIN {X 0,Y 481.746,Z 313.101,A -85,B 0,C 180,E1 -6765.223,E2 -6765.223} C_VEL
LIN {X 0,Y 481.715,Z 313.101,A -85,B 0,C 180,E1 -6768.721,E2 -6768.721} C_VEL
LIN {X 0,Y 481.65,Z 313.117,A -85,B 0,C 180,E1 -6771.394,E2 -6771.394} C_VEL
LIN {X 0,Y 481.679,Z 313.106,A -85,B 0,C 180,E1 -6774.112,E2 -6774.112} C_VEL
LIN {X 0,Y 481.748,Z 313.102,A -85,B 0,C 180,E1 -6777.138,E2 -6777.138} C_VEL
LIN {X 0,Y 481.679,Z 313.108,A -85,B 0,C 180,E1 -6779.74,E2 -6779.74} C_VEL
LIN {X 0,Y 481.673,Z 313.107,A -85,B 0,C 180,E1 -6782.673,E2 -6782.673} C_VEL
LIN {X 0,Y 481.636,Z 313.113,A -85,B 0,C 180,E1 -6785.708,E2 -6785.708} C_VEL
LIN {X 0,Y 481.67,Z 313.111,A -85,B 0,C 180,E1 -6788.858,E2 -6788.858} C_VEL
LIN {X 0,Y 481.66,Z 313.108,A -85,B 0,C 180,E1 -6791.913,E2 -6791.913} C_VEL
LIN {X 0,Y 481.657,Z 313.109,A -85,B 0,C 180,E1 -6794.456,E2 -6794.456} C_VEL
LIN {X 0,Y 481.674,Z 313.112,A -85,B 0,C 180,E1 -6796.846,E2 -6796.846} C_VEL
LIN {X 0,Y 481.673,Z 313.106,A -85,B 0,C 180,E1 -6800.059,E2 -6800.059} C_VEL
LIN {X 0,Y 481.625,Z 313.116,A -85,B 0,C 180,E1 -6803.253,E2 -6803.253} C_VEL
LIN {X 0,Y 481.704,Z 313.104,A -85,B 0,C 180,E1 -6806.329,E2 -6806.329} C_VEL
LIN {X 0,Y 481.659,Z 313.109,A -85,B 0,C 180,E1 -6809.414,E2 -6809.414} C_VEL
LIN {X 0,Y 481.697,Z 313.104,A -85,B 0,C 180,E1 -6812.167,E2 -6812.167} C_VEL
LIN {X 0,Y 481.712,Z 313.107,A -85,B 0,C 180,E1 -6814.969,E2 -6814.969} C_VEL
LIN {X 0,Y 481.646,Z 313.109,A -85,B 0,C 180,E1 -6817.704,E2 -6817.704} C_VEL
LIN {X 0,Y 481.701,Z 313.107,A -85,B 0,C 180,E1 -6820.393,E2 -6820.393} C_VEL
LIN {X 0,Y 481.686,Z 313.108,A -85,B 0,C 180,E1 -6823.033,E2 -6823.033} C_VEL
LIN {X 0,Y 481.683,Z 313.105,A -85,B 0,C 180,E1 -6825.638,E2 -6825.638} C_VEL
LIN {X 0,Y 481.743,Z 313.101,A -85,B 0,C 180,E1 -6828.215,E2 -6828.215} C_VEL
LIN {X 0,Y 481.756,Z 313.096,A -85,B 0,C 180,E1 -6831.611,E2 -6831.611} C_VEL
LIN {X 0,Y 481.81,Z 313.093,A -85,B 0,C 180,E1 -6834.139,E2 -6834.139} C_VEL
LIN {X 0,Y 481.922,Z 313.075,A -85,B 0,C 180,E1 -6837.492,E2 -6837.492} C_VEL
LIN {X 0,Y 481.918,Z 313.078,A -85,B 0,C 180,E1 -6840.835,E2 -6840.835} C_VEL
LIN {X 0,Y 481.921,Z 313.081,A -85,B 0,C 180,E1 -6842.507,E2 -6842.507} C_VEL
LIN {X 0,Y 481.809,Z 313.092,A -85,B 0,C 180,E1 -6845.86,E2 -6845.86} C_VEL
LIN {X 0,Y 481.755,Z 313.102,A -85,B 0,C 180,E1 -6848.388,E2 -6848.388} C_VEL
LIN {X 0,Y 481.787,Z 313.095,A -85,B 0,C 180,E1 -6851.784,E2 -6851.784} C_VEL
LIN {X 0,Y 481.734,Z 313.098,A -85,B 0,C 180,E1 -6855.224,E2 -6855.224} C_VEL
LIN {X 0,Y 481.704,Z 313.103,A -85,B 0,C 180,E1 -6858.722,E2 -6858.722} C_VEL
LIN {X 0,Y 481.638,Z 313.111,A -85,B 0,C 180,E1 -6861.395,E2 -6861.395} C_VEL
LIN {X 0,Y 481.67,Z 313.114,A -85,B 0,C 180,E1 -6864.113,E2 -6864.113} C_VEL
LIN {X 0,Y 481.739,Z 313.098,A -85,B 0,C 180,E1 -6867.14,E2 -6867.14} C_VEL
LIN {X 0,Y 481.681,Z 313.111,A -85,B 0,C 180,E1 -6869.741,E2 -6869.741} C_VEL
LIN {X 0,Y 481.666,Z 313.107,A -85,B 0,C 180,E1 -6872.675,E2 -6872.675} C_VEL
LIN {X 0,Y 481.636,Z 313.117,A -85,B 0,C 180,E1 -6875.709,E2 -6875.709} C_VEL
LIN {X 0,Y 481.713,Z 313.106,A -85,B 0,C 180,E1 -6879.355,E2 -6879.355} C_VEL
LIN {X 0,Y 481.643,Z 313.116,A -85,B 0,C 180,E1 -6882.161,E2 -6882.161} C_VEL
LIN {X 0,Y 481.655,Z 313.116,A -85,B 0,C 180,E1 -6885.544,E2 -6885.544} C_VEL
LIN {X 0,Y 481.69,Z 313.268,A -85,B 0,C 180,E1 -6886.077,E2 -6886.077} C_VEL
LIN {X 0,Y 483.912,Z 323.755,A -85,B 0,C 180,E1 -6889.192,E2 -6889.192} C_VEL
LIN {X 0,Y 484.889,Z 329.891,A -85,B 0,C 180,E1 -6890.915,E2 -6890.915} C_VEL
LIN {X 0,Y 484.434,Z 338.7,A -85,B 0,C 180,E1 -6893.208,E2 -6893.208} C_VEL
LIN {X 0,Y 483.722,Z 351.723,A -85,B 0,C 180,E1 -6896.49,E2 -6896.49} C_VEL
LIN {X 0,Y 483.198,Z 365.571,A -85,B 0,C 180,E1 -6899.882,E2 -6899.882} C_VEL
LIN {X 0,Y 482.678,Z 379.395,A -85,B 0,C 180,E1 -6903.169,E2 -6903.169} C_VEL
LIN {X 0,Y 482.321,Z 393.003,A -85,B 0,C 180,E1 -6906.33,E2 -6906.33} C_VEL
LIN {X 0,Y 481.872,Z 408.955,A -85,B 0,C 180,E1 -6909.957,E2 -6909.957} C_VEL
LIN {X 0,Y 481.672,Z 417.751,A -85,B 0,C 180,E1 -6911.891,E2 -6911.891} C_VEL
LIN {X 0,Y 482.236,Z 421.797,A -85,B 0,C 180,E1 -6912.038,E2 -6912.038} C_VEL
LIN {X 0,Y 484.267,Z 436.698,A -85,B 0,C 180,E1 -6912.475,E2 -6912.475} C_VEL
LIN {X 0,Y 485.013,Z 441.866,A -85,B 0,C 180,E1 -6912.666,E2 -6912.666} C_VEL
LIN {X 0,Y 484.461,Z 455.836,A -85,B 0,C 180,E1 -6913.226,E2 -6913.226} C_VEL
LIN {X 0,Y 483.883,Z 469.937,A -85,B 0,C 180,E1 -6913.982,E2 -6913.982} C_VEL
LIN {X 0,Y 483.275,Z 482.401,A -85,B 0,C 180,E1 -6914.826,E2 -6914.826} C_VEL
LIN {X 0,Y 482.736,Z 495.078,A -85,B 0,C 180,E1 -6915.887,E2 -6915.887} C_VEL
LIN {X 0,Y 482.229,Z 505.494,A -85,B 0,C 180,E1 -6916.945,E2 -6916.945} C_VEL
LIN {X 0,Y 481.843,Z 515.908,A -85,B 0,C 180,E1 -6918.218,E2 -6918.218} C_VEL
LIN {X 0,Y 481.523,Z 524.546,A -85,B 0,C 180,E1 -6919.489,E2 -6919.489} C_VEL
LIN {X 0,Y 481.264,Z 532.811,A -85,B 0,C 180,E1 -6920.969,E2 -6920.969} C_VEL
LIN {X 0,Y 481.118,Z 539.477,A -85,B 0,C 180,E1 -6922.446,E2 -6922.446} C_VEL
LIN {X 0,Y 481.112,Z 543.92,A -85,B 0,C 180,E1 -6923.657,E2 -6923.657} C_VEL
LIN {X 0,Y 481.054,Z 547.714,A -85,B 0,C 180,E1 -6924.972,E2 -6924.972} C_VEL
LIN {X 0,Y 481.035,Z 551.223,A -85,B 0,C 180,E1 -6926.65,E2 -6926.65} C_VEL
LIN {X 0,Y 480.98,Z 553.265,A -85,B 0,C 180,E1 -6928.326,E2 -6928.326} C_VEL
LIN {X 0,Y 481.043,Z 553.906,A -85,B 0,C 180,E1 -6930.001,E2 -6930.001} C_VEL
LIN {X 0,Y 481.058,Z 553.693,A -85,B 0,C 180,E1 -6930.838,E2 -6930.838} C_VEL
LIN {X 0,Y 481.052,Z 552.194,A -85,B 0,C 180,E1 -6932.513,E2 -6932.513} C_VEL
LIN {X 0,Y 481.127,Z 549.262,A -85,B 0,C 180,E1 -6934.189,E2 -6934.189} C_VEL
LIN {X 0,Y 481.112,Z 544.774,A -85,B 0,C 180,E1 -6935.87,E2 -6935.87} C_VEL
LIN {X 0,Y 481.158,Z 540.337,A -85,B 0,C 180,E1 -6937.133,E2 -6937.133} C_VEL
LIN {X 0,Y 481.264,Z 533.842,A -85,B 0,C 180,E1 -6938.609,E2 -6938.609} C_VEL
LIN {X 0,Y 481.407,Z 525.729,A -85,B 0,C 180,E1 -6940.09,E2 -6940.09} C_VEL
LIN {X 0,Y 481.721,Z 517.295,A -85,B 0,C 180,E1 -6941.36,E2 -6941.36} C_VEL
LIN {X 0,Y 482.045,Z 507.129,A -85,B 0,C 180,E1 -6942.633,E2 -6942.633} C_VEL
LIN {X 0,Y 482.459,Z 495.91,A -85,B 0,C 180,E1 -6943.801,E2 -6943.801} C_VEL
LIN {X 0,Y 483.018,Z 483.592,A -85,B 0,C 180,E1 -6944.86,E2 -6944.86} C_VEL
LIN {X 0,Y 483.575,Z 469.975,A -85,B 0,C 180,E1 -6945.814,E2 -6945.814} C_VEL
LIN {X 0,Y 484.204,Z 455.378,A -85,B 0,C 180,E1 -6946.614,E2 -6946.614} C_VEL
LIN {X 0,Y 484.625,Z 440.373,A -85,B 0,C 180,E1 -6947.241,E2 -6947.241} C_VEL
LIN {X 0,Y 483.055,Z 428.511,A -85,B 0,C 180,E1 -6947.668,E2 -6947.668} C_VEL
LIN {X 0,Y 481.615,Z 413.778,A -85,B 0,C 180,E1 -6948.081,E2 -6948.081} C_VEL
LIN {X 0,Y 481.595,Z 410.383,A -85,B 0,C 180,E1 -6948.727,E2 -6948.727} C_VEL
LIN {X 0,Y 481.753,Z 397.623,A -85,B 0,C 180,E1 -6951.39,E2 -6951.39} C_VEL
LIN {X 0,Y 481.89,Z 383.686,A -85,B 0,C 180,E1 -6954.331,E2 -6954.331} C_VEL
LIN {X 0,Y 482.032,Z 369.14,A -85,B 0,C 180,E1 -6957.464,E2 -6957.464} C_VEL
LIN {X 0,Y 482.105,Z 356.826,A -85,B 0,C 180,E1 -6960.195,E2 -6960.195} C_VEL
LIN {X 0,Y 482.23,Z 345.205,A -85,B 0,C 180,E1 -6962.881,E2 -6962.881} C_VEL
LIN {X 0,Y 482.78,Z 331.959,A -85,B 0,C 180,E1 -6966.127,E2 -6966.127} C_VEL
LIN {X 0,Y 483.411,Z 323.831,A -85,B 0,C 180,E1 -6968.273,E2 -6968.273} C_VEL
LIN {X 0,Y 482.974,Z 319.583,A -85,B 0,C 180,E1 -6969.536,E2 -6969.536} C_VEL
LIN {X 0,Y 481.694,Z 313.177,A -85,B 0,C 180,E1 -6971.713,E2 -6971.713} C_VEL
LIN {X 0,Y 481.663,Z 313.113,A -85,B 0,C 180,E1 -6974.458,E2 -6974.458} C_VEL
LIN {X 0,Y 481.652,Z 313.116,A -85,B 0,C 180,E1 -6977.84,E2 -6977.84} C_VEL
LIN {X 0,Y 481.718,Z 313.104,A -85,B 0,C 180,E1 -6980.646,E2 -6980.646} C_VEL
LIN {X 0,Y 481.647,Z 313.112,A -85,B 0,C 180,E1 -6984.291,E2 -6984.291} C_VEL
LIN {X 0,Y 481.676,Z 313.112,A -85,B 0,C 180,E1 -6987.326,E2 -6987.326} C_VEL
LIN {X 0,Y 481.682,Z 313.107,A -85,B 0,C 180,E1 -6990.259,E2 -6990.259} C_VEL
LIN {X 0,Y 481.749,Z 313.103,A -85,B 0,C 180,E1 -6993.112,E2 -6993.112} C_VEL
LIN {X 0,Y 481.681,Z 313.11,A -85,B 0,C 180,E1 -6995.887,E2 -6995.887} C_VEL
LIN {X 0,Y 481.706,Z 313.11,A -85,B 0,C 180,E1 -6999.028,E2 -6999.028} C_VEL
LIN {X 0,Y 481.761,Z 313.313,A -85,B 0,C 180,E1 -7001.688,E2 -7001.688} C_VEL
LIN {X 0,Y 482.152,Z 314.729,A -85,B 0,C 180,E1 -7001.857,E2 -7001.857} C_VEL
LIN {X 0,Y 485.411,Z 325.442,A -85,B 0,C 180,E1 -7002.517,E2 -7002.517} C_VEL
LIN {X 0,Y 484.937,Z 337.938,A -85,B 0,C 180,E1 -7003.238,E2 -7003.238} C_VEL
LIN {X 0,Y 484.464,Z 349.943,A -85,B 0,C 180,E1 -7004.109,E2 -7004.109} C_VEL
LIN {X 0,Y 483.976,Z 360.698,A -85,B 0,C 180,E1 -7005.063,E2 -7005.063} C_VEL
LIN {X 0,Y 483.471,Z 370.637,A -85,B 0,C 180,E1 -7006.122,E2 -7006.122} C_VEL
LIN {X 0,Y 482.919,Z 380.49,A -85,B 0,C 180,E1 -7007.391,E2 -7007.391} C_VEL
LIN {X 0,Y 482.571,Z 388.587,A -85,B 0,C 180,E1 -7008.661,E2 -7008.661} C_VEL
LIN {X 0,Y 482.201,Z 395.315,A -85,B 0,C 180,E1 -7009.927,E2 -7009.927} C_VEL
LIN {X 0,Y 481.941,Z 400.836,A -85,B 0,C 180,E1 -7011.193,E2 -7011.193} C_VEL
LIN {X 0,Y 481.674,Z 406.531,A -85,B 0,C 180,E1 -7012.829,E2 -7012.829} C_VEL
LIN {X 0,Y 481.528,Z 409.948,A -85,B 0,C 180,E1 -7014.136,E2 -7014.136} C_VEL
LIN {X 0,Y 481.346,Z 413.09,A -85,B 0,C 180,E1 -7015.814,E2 -7015.814} C_VEL
LIN {X 0,Y 481.224,Z 414.855,A -85,B 0,C 180,E1 -7017.489,E2 -7017.489} C_VEL
LIN {X 0,Y 481.183,Z 415.284,A -85,B 0,C 180,E1 -7019.163,E2 -7019.163} C_VEL
LIN {X 0,Y 481.186,Z 414.403,A -85,B 0,C 180,E1 -7020.837,E2 -7020.837} C_VEL
LIN {X 0,Y 481.219,Z 412.207,A -85,B 0,C 180,E1 -7022.511,E2 -7022.511} C_VEL
LIN {X 0,Y 481.405,Z 408.626,A -85,B 0,C 180,E1 -7024.186,E2 -7024.186} C_VEL
LIN {X 0,Y 481.537,Z 403.584,A -85,B 0,C 180,E1 -7025.864,E2 -7025.864} C_VEL
LIN {X 0,Y 481.816,Z 397.92,A -85,B 0,C 180,E1 -7027.304,E2 -7027.304} C_VEL
LIN {X 0,Y 482.143,Z 390.568,A -85,B 0,C 180,E1 -7028.804,E2 -7028.804} C_VEL
LIN {X 0,Y 482.482,Z 382.997,A -85,B 0,C 180,E1 -7030.067,E2 -7030.067} C_VEL
LIN {X 0,Y 482.876,Z 373.911,A -85,B 0,C 180,E1 -7031.332,E2 -7031.332} C_VEL
LIN {X 0,Y 483.417,Z 364.83,A -85,B 0,C 180,E1 -7032.383,E2 -7032.383} C_VEL
LIN {X 0,Y 483.931,Z 354.017,A -85,B 0,C 180,E1 -7033.437,E2 -7033.437} C_VEL
LIN {X 0,Y 484.423,Z 342.205,A -85,B 0,C 180,E1 -7034.386,E2 -7034.386} C_VEL
LIN {X 0,Y 484.926,Z 328.723,A -85,B 0,C 180,E1 -7035.255,E2 -7035.255} C_VEL
LIN {X 0,Y 484.986,Z 323.966,A -85,B 0,C 180,E1 -7035.518,E2 -7035.518} C_VEL
LIN {X 0,Y 481.809,Z 313.675,A -85,B 0,C 180,E1 -7036.172,E2 -7036.172} C_VEL
LIN {X 0,Y 481.73,Z 313.148,A -85,B 0,C 180,E1 -7036.311,E2 -7036.311} C_VEL
LIN {X 0,Y 481.71,Z 313.106,A -85,B 0,C 180,E1 -7039.607,E2 -7039.607} C_VEL
LIN {X 0,Y 481.654,Z 313.114,A -85,B 0,C 180,E1 -7042.295,E2 -7042.295} C_VEL
LIN {X 0,Y 481.715,Z 313.103,A -85,B 0,C 180,E1 -7045.236,E2 -7045.236} C_VEL
LIN {X 0,Y 481.705,Z 313.102,A -85,B 0,C 180,E1 -7047.832,E2 -7047.832} C_VEL
LIN {X 0,Y 481.651,Z 313.116,A -85,B 0,C 180,E1 -7050.711,E2 -7050.711} C_VEL
LIN {X 0,Y 481.702,Z 313.102,A -85,B 0,C 180,E1 -7053.733,E2 -7053.733} C_VEL
LIN {X 0,Y 481.634,Z 313.116,A -85,B 0,C 180,E1 -7056.747,E2 -7056.747} C_VEL
LIN {X 0,Y 481.682,Z 313.106,A -85,B 0,C 180,E1 -7059.94,E2 -7059.94} C_VEL
LIN {X 0,Y 481.638,Z 313.111,A -85,B 0,C 180,E1 -7063.147,E2 -7063.147} C_VEL
LIN {X 0,Y 481.665,Z 313.107,A -85,B 0,C 180,E1 -7065.641,E2 -7065.641} C_VEL
LIN {X 0,Y 481.669,Z 313.108,A -85,B 0,C 180,E1 -7068.959,E2 -7068.959} C_VEL
LIN {X 0,Y 481.66,Z 313.111,A -85,B 0,C 180,E1 -7071.993,E2 -7071.993} C_VEL
LIN {X 0,Y 481.694,Z 313.103,A -85,B 0,C 180,E1 -7075.318,E2 -7075.318} C_VEL
LIN {X 0,Y 481.651,Z 313.116,A -85,B 0,C 180,E1 -7078.311,E2 -7078.311} C_VEL
LIN {X 0,Y 481.706,Z 313.102,A -85,B 0,C 180,E1 -7081.218,E2 -7081.218} C_VEL
LIN {X 0,Y 481.751,Z 313.096,A -85,B 0,C 180,E1 -7083.002,E2 -7083.002} C_VEL
LIN {X 0,Y 481.092,Z 313.182,A -85,B 0,C 180,E1 -7083.699,E2 -7083.699} C_VEL
LIN {X 0,Y 478.243,Z 313.537,A -85,B 0,C 180,E1 -7084.832,E2 -7084.832} C_VEL
LIN {X 0,Y 475.81,Z 313.841,A -85,B 0,C 180,E1 -7085.745,E2 -7085.745} C_VEL
LIN {X 0,Y 474.738,Z 313.974,A -85,B 0,C 180,E1 -7086.45,E2 -7086.45} C_VEL
LIN {X 0,Y 474.636,Z 313.984,A -85,B 0,C 180,E1 -7086.689,E2 -7086.689} C_VEL
LIN {X 0,Y 474.661,Z 313.987,A -85,B 0,C 180,E1 -7090.089,E2 -7090.089} C_VEL
LIN {X 0,Y 474.657,Z 313.98,A -85,B 0,C 180,E1 -7092.774,E2 -7092.774} C_VEL
LIN {X 0,Y 474.655,Z 313.982,A -85,B 0,C 180,E1 -7095.421,E2 -7095.421} C_VEL
LIN {X 0,Y 474.711,Z 313.98,A -85,B 0,C 180,E1 -7098.037,E2 -7098.037} C_VEL
LIN {X 0,Y 474.733,Z 313.974,A -85,B 0,C 180,E1 -7101.486,E2 -7101.486} C_VEL
LIN {X 0,Y 474.776,Z 313.97,A -85,B 0,C 180,E1 -7104.052,E2 -7104.052} C_VEL
LIN {X 0,Y 474.899,Z 313.954,A -85,B 0,C 180,E1 -7107.455,E2 -7107.455} C_VEL
LIN {X 0,Y 474.917,Z 313.952,A -85,B 0,C 180,E1 -7109.999,E2 -7109.999} C_VEL
LIN {X 0,Y 474.899,Z 313.95,A -85,B 0,C 180,E1 -7112.544,E2 -7112.544} C_VEL
LIN {X 0,Y 474.783,Z 313.969,A -85,B 0,C 180,E1 -7115.947,E2 -7115.947} C_VEL
LIN {X 0,Y 474.732,Z 313.971,A -85,B 0,C 180,E1 -7118.513,E2 -7118.513} C_VEL
LIN {X 0,Y 474.708,Z 313.977,A -85,B 0,C 180,E1 -7121.961,E2 -7121.961} C_VEL
LIN {X 0,Y 474.703,Z 313.982,A -85,B 0,C 180,E1 -7125.455,E2 -7125.455} C_VEL
LIN {X 0,Y 474.668,Z 313.981,A -85,B 0,C 180,E1 -7129.009,E2 -7129.009} C_VEL
LIN {X 0,Y 474.593,Z 313.992,A -85,B 0,C 180,E1 -7131.728,E2 -7131.728} C_VEL
LIN {X 0,Y 474.661,Z 313.98,A -85,B 0,C 180,E1 -7134.492,E2 -7134.492} C_VEL
LIN {X 0,Y 474.7,Z 313.983,A -85,B 0,C 180,E1 -7137.338,E2 -7137.338} C_VEL
LIN {X 0,Y 474.605,Z 313.989,A -85,B 0,C 180,E1 -7140.809,E2 -7140.809} C_VEL
LIN {X 0,Y 474.636,Z 313.983,A -85,B 0,C 180,E1 -7143.983,E2 -7143.983} C_VEL
LIN {X 0,Y 474.571,Z 313.995,A -85,B 0,C 180,E1 -7146.898,E2 -7146.898} C_VEL
LIN {X 0,Y 474.626,Z 313.986,A -85,B 0,C 180,E1 -7149.647,E2 -7149.647} C_VEL
LIN {X 0,Y 474.633,Z 313.989,A -85,B 0,C 180,E1 -7152.931,E2 -7152.931} C_VEL
LIN {X 0,Y 474.612,Z 313.986,A -85,B 0,C 180,E1 -7155.895,E2 -7155.895} C_VEL
LIN {X 0,Y 474.624,Z 313.992,A -85,B 0,C 180,E1 -7159.04,E2 -7159.04} C_VEL
LIN {X 0,Y 474.61,Z 313.986,A -85,B 0,C 180,E1 -7161.702,E2 -7161.702} C_VEL
LIN {X 0,Y 474.625,Z 313.99,A -85,B 0,C 180,E1 -7164.725,E2 -7164.725} C_VEL
LIN {X 0,Y 474.632,Z 313.983,A -85,B 0,C 180,E1 -7167.787,E2 -7167.787} C_VEL
LIN {X 0,Y 474.627,Z 313.991,A -85,B 0,C 180,E1 -7170.882,E2 -7170.882} C_VEL
LIN {X 0,Y 474.66,Z 313.98,A -85,B 0,C 180,E1 -7173.628,E2 -7173.628} C_VEL
LIN {X 0,Y 474.629,Z 313.99,A -85,B 0,C 180,E1 -7176.64,E2 -7176.64} C_VEL
LIN {X 0,Y 474.65,Z 313.982,A -85,B 0,C 180,E1 -7180.089,E2 -7180.089} C_VEL
LIN {X 0,Y 474.645,Z 313.988,A -85,B 0,C 180,E1 -7182.774,E2 -7182.774} C_VEL
LIN {X 0,Y 474.641,Z 313.982,A -85,B 0,C 180,E1 -7185.42,E2 -7185.42} C_VEL
LIN {X 0,Y 474.696,Z 313.977,A -85,B 0,C 180,E1 -7188.037,E2 -7188.037} C_VEL
LIN {X 0,Y 474.721,Z 313.972,A -85,B 0,C 180,E1 -7191.486,E2 -7191.486} C_VEL
LIN {X 0,Y 474.772,Z 313.968,A -85,B 0,C 180,E1 -7194.052,E2 -7194.052} C_VEL
LIN {X 0,Y 474.888,Z 313.951,A -85,B 0,C 180,E1 -7197.455,E2 -7197.455} C_VEL
LIN {X 0,Y 474.869,Z 313.956,A -85,B 0,C 180,E1 -7200.848,E2 -7200.848} C_VEL
LIN {X 0,Y 474.887,Z 313.957,A -85,B 0,C 180,E1 -7202.544,E2 -7202.544} C_VEL
LIN {X 0,Y 474.771,Z 313.969,A -85,B 0,C 180,E1 -7205.947,E2 -7205.947} C_VEL
LIN {X 0,Y 474.72,Z 313.977,A -85,B 0,C 180,E1 -7208.513,E2 -7208.513} C_VEL
LIN {X 0,Y 474.73,Z 313.976,A -85,B 0,C 180,E1 -7211.962,E2 -7211.962} C_VEL
LIN {X 0,Y 474.693,Z 313.979,A -85,B 0,C 180,E1 -7215.777,E2 -7215.777} C_VEL
LIN {X 0,Y 474.657,Z 313.98,A -85,B 0,C 180,E1 -7219.01,E2 -7219.01} C_VEL
LIN {X 0,Y 474.583,Z 313.993,A -85,B 0,C 180,E1 -7221.729,E2 -7221.729} C_VEL
LIN {X 0,Y 474.651,Z 313.983,A -85,B 0,C 180,E1 -7224.493,E2 -7224.493} C_VEL
LIN {X 0,Y 474.691,Z 313.977,A -85,B 0,C 180,E1 -7227.339,E2 -7227.339} C_VEL
LIN {X 0,Y 474.603,Z 313.987,A -85,B 0,C 180,E1 -7230.812,E2 -7230.812} C_VEL
LIN {X 0,Y 474.631,Z 313.99,A -85,B 0,C 180,E1 -7233.985,E2 -7233.985} C_VEL
LIN {X 0,Y 474.57,Z 313.993,A -85,B 0,C 180,E1 -7236.901,E2 -7236.901} C_VEL
LIN {X 0,Y 474.649,Z 313.989,A -85,B 0,C 180,E1 -7239.652,E2 -7239.652} C_VEL
LIN {X 0,Y 474.609,Z 313.991,A -85,B 0,C 180,E1 -7242.935,E2 -7242.935} C_VEL
LIN {X 0,Y 474.64,Z 314.097,A -85,B 0,C 180,E1 -7245.717,E2 -7245.717} C_VEL
LIN {X 0,Y 476.767,Z 324.063,A -85,B 0,C 180,E1 -7248.745,E2 -7248.745} C_VEL
LIN {X 0,Y 477.961,Z 331.152,A -85,B 0,C 180,E1 -7250.783,E2 -7250.783} C_VEL
LIN {X 0,Y 477.562,Z 339.129,A -85,B 0,C 180,E1 -7252.889,E2 -7252.889} C_VEL
LIN {X 0,Y 476.854,Z 351.015,A -85,B 0,C 180,E1 -7255.942,E2 -7255.942} C_VEL
LIN {X 0,Y 476.278,Z 364.865,A -85,B 0,C 180,E1 -7259.398,E2 -7259.398} C_VEL
LIN {X 0,Y 475.74,Z 378.661,A -85,B 0,C 180,E1 -7262.746,E2 -7262.746} C_VEL
LIN {X 0,Y 475.28,Z 392.445,A -85,B 0,C 180,E1 -7266.007,E2 -7266.007} C_VEL
LIN {X 0,Y 474.864,Z 406.2,A -85,B 0,C 180,E1 -7269.195,E2 -7269.195} C_VEL
LIN {X 0,Y 474.615,Z 416.958,A -85,B 0,C 180,E1 -7271.62,E2 -7271.62} C_VEL
LIN {X 0,Y 474.988,Z 419.912,A -85,B 0,C 180,E1 -7271.742,E2 -7271.742} C_VEL
LIN {X 0,Y 477.011,Z 435.037,A -85,B 0,C 180,E1 -7272.186,E2 -7272.186} C_VEL
LIN {X 0,Y 478.085,Z 442.915,A -85,B 0,C 180,E1 -7272.489,E2 -7272.489} C_VEL
LIN {X 0,Y 477.539,Z 456.415,A -85,B 0,C 180,E1 -7273.061,E2 -7273.061} C_VEL
LIN {X 0,Y 477.005,Z 468.846,A -85,B 0,C 180,E1 -7273.744,E2 -7273.744} C_VEL
LIN {X 0,Y 476.356,Z 481.328,A -85,B 0,C 180,E1 -7274.6,E2 -7274.6} C_VEL
LIN {X 0,Y 475.733,Z 494.015,A -85,B 0,C 180,E1 -7275.674,E2 -7275.674} C_VEL
LIN {X 0,Y 475.21,Z 504.45,A -85,B 0,C 180,E1 -7276.749,E2 -7276.749} C_VEL
LIN {X 0,Y 474.796,Z 514.888,A -85,B 0,C 180,E1 -7278.041,E2 -7278.041} C_VEL
LIN {X 0,Y 474.46,Z 523.539,A -85,B 0,C 180,E1 -7279.331,E2 -7279.331} C_VEL
LIN {X 0,Y 474.2,Z 531.817,A -85,B 0,C 180,E1 -7280.833,E2 -7280.833} C_VEL
LIN {X 0,Y 474.04,Z 538.488,A -85,B 0,C 180,E1 -7282.333,E2 -7282.333} C_VEL
LIN {X 0,Y 474.036,Z 544.403,A -85,B 0,C 180,E1 -7284.044,E2 -7284.044} C_VEL
LIN {X 0,Y 473.99,Z 548.674,A -85,B 0,C 180,E1 -7285.749,E2 -7285.749} C_VEL
LIN {X 0,Y 473.983,Z 551.44,A -85,B 0,C 180,E1 -7287.451,E2 -7287.451} C_VEL
LIN {X 0,Y 473.927,Z 552.76,A -85,B 0,C 180,E1 -7289.151,E2 -7289.151} C_VEL
LIN {X 0,Y 474.03,Z 552.907,A -85,B 0,C 180,E1 -7290.001,E2 -7290.001} C_VEL
LIN {X 0,Y 474.047,Z 552.684,A -85,B 0,C 180,E1 -7290.85,E2 -7290.85} C_VEL
LIN {X 0,Y 474.017,Z 551.157,A -85,B 0,C 180,E1 -7292.55,E2 -7292.55} C_VEL
LIN {X 0,Y 474.099,Z 548.193,A -85,B 0,C 180,E1 -7294.251,E2 -7294.251} C_VEL
LIN {X 0,Y 474.089,Z 544.951,A -85,B 0,C 180,E1 -7295.53,E2 -7295.53} C_VEL
LIN {X 0,Y 474.096,Z 540.767,A -85,B 0,C 180,E1 -7296.812,E2 -7296.812} C_VEL
LIN {X 0,Y 474.162,Z 535.614,A -85,B 0,C 180,E1 -7298.095,E2 -7298.095} C_VEL
LIN {X 0,Y 474.309,Z 528.169,A -85,B 0,C 180,E1 -7299.596,E2 -7299.596} C_VEL
LIN {X 0,Y 474.539,Z 518.965,A -85,B 0,C 180,E1 -7301.101,E2 -7301.101} C_VEL
LIN {X 0,Y 474.849,Z 509.664,A -85,B 0,C 180,E1 -7302.357,E2 -7302.357} C_VEL
LIN {X 0,Y 475.342,Z 497.816,A -85,B 0,C 180,E1 -7303.684,E2 -7303.684} C_VEL
LIN {X 0,Y 475.855,Z 486.146,A -85,B 0,C 180,E1 -7304.761,E2 -7304.761} C_VEL
LIN {X 0,Y 476.457,Z 473.381,A -85,B 0,C 180,E1 -7305.727,E2 -7305.727} C_VEL
LIN {X 0,Y 477.037,Z 460.496,A -85,B 0,C 180,E1 -7306.519,E2 -7306.519} C_VEL
LIN {X 0,Y 477.618,Z 445.851,A -85,B 0,C 180,E1 -7307.226,E2 -7307.226} C_VEL
LIN {X 0,Y 477.577,Z 440.434,A -85,B 0,C 180,E1 -7307.448,E2 -7307.448} C_VEL
LIN {X 0,Y 476.248,Z 429.371,A -85,B 0,C 180,E1 -7307.873,E2 -7307.873} C_VEL
LIN {X 0,Y 474.514,Z 412.416,A -85,B 0,C 180,E1 -7308.37,E2 -7308.37} C_VEL
LIN {X 0,Y 474.524,Z 410.326,A -85,B 0,C 180,E1 -7308.747,E2 -7308.747} C_VEL
LIN {X 0,Y 474.687,Z 396.31,A -85,B 0,C 180,E1 -7311.725,E2 -7311.725} C_VEL
LIN {X 0,Y 474.826,Z 381.334,A -85,B 0,C 180,E1 -7314.951,E2 -7314.951} C_VEL
LIN {X 0,Y 475.021,Z 366.359,A -85,B 0,C 180,E1 -7318.259,E2 -7318.259} C_VEL
LIN {X 0,Y 475.211,Z 352.576,A -85,B 0,C 180,E1 -7321.421,E2 -7321.421} C_VEL
LIN {X 0,Y 475.577,Z 337.132,A -85,B 0,C 180,E1 -7325.194,E2 -7325.194} C_VEL
LIN {X 0,Y 476.505,Z 325.534,A -85,B 0,C 180,E1 -7328.277,E2 -7328.277} C_VEL
LIN {X 0,Y 476.206,Z 321.835,A -85,B 0,C 180,E1 -7329.391,E2 -7329.391} C_VEL
LIN {X 0,Y 474.685,Z 314.275,A -85,B 0,C 180,E1 -7332.005,E2 -7332.005} C_VEL
LIN {X 0,Y 474.634,Z 313.998,A -85,B 0,C 180,E1 -7332.238,E2 -7332.238} C_VEL
LIN {X 0,Y 474.624,Z 313.992,A -85,B 0,C 180,E1 -7335.297,E2 -7335.297} C_VEL
LIN {X 0,Y 474.627,Z 313.989,A -85,B 0,C 180,E1 -7338.215,E2 -7338.215} C_VEL
LIN {X 0,Y 474.672,Z 313.982,A -85,B 0,C 180,E1 -7340.457,E2 -7340.457} C_VEL
LIN {X 0,Y 474.597,Z 313.995,A -85,B 0,C 180,E1 -7343.677,E2 -7343.677} C_VEL
LIN {X 0,Y 474.646,Z 313.986,A -85,B 0,C 180,E1 -7346.78,E2 -7346.78} C_VEL
LIN {X 0,Y 474.609,Z 313.991,A -85,B 0,C 180,E1 -7349.77,E2 -7349.77} C_VEL
LIN {X 0,Y 474.7,Z 313.979,A -85,B 0,C 180,E1 -7352.68,E2 -7352.68} C_VEL
LIN {X 0,Y 474.663,Z 313.987,A -85,B 0,C 180,E1 -7355.507,E2 -7355.507} C_VEL
LIN {X 0,Y 474.674,Z 313.986,A -85,B 0,C 180,E1 -7359.186,E2 -7359.186} C_VEL
LIN {X 0,Y 474.685,Z 314.107,A -85,B 0,C 180,E1 -7361.363,E2 -7361.363} C_VEL
LIN {X 0,Y 474.931,Z 315.194,A -85,B 0,C 180,E1 -7361.53,E2 -7361.53} C_VEL
LIN {X 0,Y 478.607,Z 326.492,A -85,B 0,C 180,E1 -7362.26,E2 -7362.26} C_VEL
LIN {X 0,Y 478.211,Z 339.009,A -85,B 0,C 180,E1 -7362.999,E2 -7362.999} C_VEL
LIN {X 0,Y 477.721,Z 350.935,A -85,B 0,C 180,E1 -7363.878,E2 -7363.878} C_VEL
LIN {X 0,Y 477.208,Z 361.697,A -85,B 0,C 180,E1 -7364.846,E2 -7364.846} C_VEL
LIN {X 0,Y 476.65,Z 371.642,A -85,B 0,C 180,E1 -7365.92,E2 -7365.92} C_VEL
LIN {X 0,Y 476.068,Z 381.511,A -85,B 0,C 180,E1 -7367.207,E2 -7367.207} C_VEL
LIN {X 0,Y 475.688,Z 389.61,A -85,B 0,C 180,E1 -7368.495,E2 -7368.495} C_VEL
LIN {X 0,Y 475.284,Z 396.344,A -85,B 0,C 180,E1 -7369.779,E2 -7369.779} C_VEL
LIN {X 0,Y 474.994,Z 401.866,A -85,B 0,C 180,E1 -7371.063,E2 -7371.063} C_VEL
LIN {X 0,Y 474.704,Z 407.559,A -85,B 0,C 180,E1 -7372.722,E2 -7372.722} C_VEL
LIN {X 0,Y 474.561,Z 410.976,A -85,B 0,C 180,E1 -7374.05,E2 -7374.05} C_VEL
LIN {X 0,Y 474.335,Z 414.124,A -85,B 0,C 180,E1 -7375.752,E2 -7375.752} C_VEL
LIN {X 0,Y 474.205,Z 415.891,A -85,B 0,C 180,E1 -7377.452,E2 -7377.452} C_VEL
LIN {X 0,Y 474.165,Z 416.313,A -85,B 0,C 180,E1 -7379.151,E2 -7379.151} C_VEL
LIN {X 0,Y 474.167,Z 415.419,A -85,B 0,C 180,E1 -7380.849,E2 -7380.849} C_VEL
LIN {X 0,Y 474.198,Z 413.208,A -85,B 0,C 180,E1 -7382.549,E2 -7382.549} C_VEL
LIN {X 0,Y 474.393,Z 409.608,A -85,B 0,C 180,E1 -7384.248,E2 -7384.248} C_VEL
LIN {X 0,Y 474.544,Z 404.54,A -85,B 0,C 180,E1 -7385.951,E2 -7385.951} C_VEL
LIN {X 0,Y 474.846,Z 398.851,A -85,B 0,C 180,E1 -7387.411,E2 -7387.411} C_VEL
LIN {X 0,Y 475.197,Z 391.468,A -85,B 0,C 180,E1 -7388.934,E2 -7388.934} C_VEL
LIN {X 0,Y 475.555,Z 383.871,A -85,B 0,C 180,E1 -7390.215,E2 -7390.215} C_VEL
LIN {X 0,Y 475.973,Z 374.756,A -85,B 0,C 180,E1 -7391.498,E2 -7391.498} C_VEL
LIN {X 0,Y 476.546,Z 365.65,A -85,B 0,C 180,E1 -7392.564,E2 -7392.564} C_VEL
LIN {X 0,Y 477.092,Z 354.813,A -85,B 0,C 180,E1 -7393.633,E2 -7393.633} C_VEL
LIN {X 0,Y 477.585,Z 342.987,A -85,B 0,C 180,E1 -7394.597,E2 -7394.597} C_VEL
LIN {X 0,Y 478.137,Z 329.768,A -85,B 0,C 180,E1 -7395.46,E2 -7395.46} C_VEL
LIN {X 0,Y 478.181,Z 325.602,A -85,B 0,C 180,E1 -7395.695,E2 -7395.695} C_VEL
LIN {X 0,Y 474.806,Z 314.735,A -85,B 0,C 180,E1 -7396.389,E2 -7396.389} C_VEL
LIN {X 0,Y 474.657,Z 314.025,A -85,B 0,C 180,E1 -7396.561,E2 -7396.561} C_VEL
LIN {X 0,Y 474.67,Z 313.987,A -85,B 0,C 180,E1 -7399.01,E2 -7399.01} C_VEL
LIN {X 0,Y 474.593,Z 313.991,A -85,B 0,C 180,E1 -7401.729,E2 -7401.729} C_VEL
LIN {X 0,Y 474.662,Z 313.986,A -85,B 0,C 180,E1 -7404.493,E2 -7404.493} C_VEL
LIN {X 0,Y 474.686,Z 313.977,A -85,B 0,C 180,E1 -7407.334,E2 -7407.334} C_VEL
LIN {X 0,Y 474.61,Z 313.989,A -85,B 0,C 180,E1 -7410.23,E2 -7410.23} C_VEL
LIN {X 0,Y 474.648,Z 313.982,A -85,B 0,C 180,E1 -7413.22,E2 -7413.22} C_VEL
LIN {X 0,Y 474.598,Z 313.992,A -85,B 0,C 180,E1 -7416.323,E2 -7416.323} C_VEL
LIN {X 0,Y 474.623,Z 313.984,A -85,B 0,C 180,E1 -7419.646,E2 -7419.646} C_VEL
LIN {X 0,Y 474.629,Z 313.989,A -85,B 0,C 180,E1 -7422.237,E2 -7422.237} C_VEL
LIN {X 0,Y 474.627,Z 313.984,A -85,B 0,C 180,E1 -7425.297,E2 -7425.297} C_VEL
LIN {X 0,Y 474.635,Z 313.989,A -85,B 0,C 180,E1 -7428.216,E2 -7428.216} C_VEL
LIN {X 0,Y 474.65,Z 313.988,A -85,B 0,C 180,E1 -7430.454,E2 -7430.454} C_VEL
LIN {X 0,Y 474.595,Z 313.989,A -85,B 0,C 180,E1 -7433.676,E2 -7433.676} C_VEL
LIN {X 0,Y 474.649,Z 313.983,A -85,B 0,C 180,E1 -7436.78,E2 -7436.78} C_VEL
LIN {X 0,Y 474.611,Z 313.988,A -85,B 0,C 180,E1 -7439.77,E2 -7439.77} C_VEL
LIN {X 0,Y 474.675,Z 313.978,A -85,B 0,C 180,E1 -7442.995,E2 -7442.995} C_VEL
LIN {X 0,Y 474.647,Z 313.982,A -85,B 0,C 180,E1 -7445.506,E2 -7445.506} C_VEL
LIN {X 0,Y 474.636,Z 313.984,A -85,B 0,C 180,E1 -7446.689,E2 -7446.689} C_VEL
LIN {X 0,Y 473.932,Z 314.072,A -85,B 0,C 180,E1 -7447.397,E2 -7447.397} C_VEL
LIN {X 0,Y 471.075,Z 314.428,A -85,B 0,C 180,E1 -7448.547,E2 -7448.547} C_VEL
LIN {X 0,Y 468.695,Z 314.724,A -85,B 0,C 180,E1 -7449.475,E2 -7449.475} C_VEL
LIN {X 0,Y 467.691,Z 314.854,A -85,B 0,C 180,E1 -7450.191,E2 -7450.191} C_VEL
LIN {X 0,Y 467.618,Z 314.857,A -85,B 0,C 180,E1 -7450.433,E2 -7450.433} C_VEL
LIN {X 0,Y 467.604,Z 314.86,A -85,B 0,C 180,E1 -7453.407,E2 -7453.407} C_VEL
LIN {X 0,Y 467.617,Z 314.863,A -85,B 0,C 180,E1 -7456.085,E2 -7456.085} C_VEL
LIN {X 0,Y 467.658,Z 314.852,A -85,B 0,C 180,E1 -7458.733,E2 -7458.733} C_VEL
LIN {X 0,Y 467.755,Z 314.843,A -85,B 0,C 180,E1 -7462.228,E2 -7462.228} C_VEL
LIN {X 0,Y 467.727,Z 314.843,A -85,B 0,C 180,E1 -7464.827,E2 -7464.827} C_VEL
LIN {X 0,Y 467.865,Z 314.829,A -85,B 0,C 180,E1 -7467.416,E2 -7467.416} C_VEL
LIN {X 0,Y 467.888,Z 314.828,A -85,B 0,C 180,E1 -7469.999,E2 -7469.999} C_VEL
LIN {X 0,Y 467.864,Z 314.826,A -85,B 0,C 180,E1 -7472.582,E2 -7472.582} C_VEL
LIN {X 0,Y 467.748,Z 314.844,A -85,B 0,C 180,E1 -7476.036,E2 -7476.036} C_VEL
LIN {X 0,Y 467.686,Z 314.848,A -85,B 0,C 180,E1 -7478.642,E2 -7478.642} C_VEL
LIN {X 0,Y 467.66,Z 314.853,A -85,B 0,C 180,E1 -7482.144,E2 -7482.144} C_VEL
LIN {X 0,Y 467.642,Z 314.859,A -85,B 0,C 180,E1 -7485.694,E2 -7485.694} C_VEL
LIN {X 0,Y 467.62,Z 314.857,A -85,B 0,C 180,E1 -7488.764,E2 -7488.764} C_VEL
LIN {X 0,Y 467.583,Z 314.867,A -85,B 0,C 180,E1 -7491.267,E2 -7491.267} C_VEL
LIN {X 0,Y 467.575,Z 314.864,A -85,B 0,C 180,E1 -7493.942,E2 -7493.942} C_VEL
LIN {X 0,Y 467.617,Z 314.859,A -85,B 0,C 180,E1 -7496.799,E2 -7496.799} C_VEL
LIN {X 0,Y 467.555,Z 314.867,A -85,B 0,C 180,E1 -7499.737,E2 -7499.737} C_VEL
LIN {X 0,Y 467.583,Z 314.863,A -85,B 0,C 180,E1 -7502.757,E2 -7502.757} C_VEL
LIN {X 0,Y 467.552,Z 314.866,A -85,B 0,C 180,E1 -7505.888,E2 -7505.888} C_VEL
LIN {X 0,Y 467.58,Z 314.87,A -85,B 0,C 180,E1 -7509.144,E2 -7509.144} C_VEL
LIN {X 0,Y 467.583,Z 314.863,A -85,B 0,C 180,E1 -7512.566,E2 -7512.566} C_VEL
LIN {X 0,Y 467.568,Z 314.871,A -85,B 0,C 180,E1 -7515.052,E2 -7515.052} C_VEL
LIN {X 0,Y 467.585,Z 314.864,A -85,B 0,C 180,E1 -7517.439,E2 -7517.439} C_VEL
LIN {X 0,Y 467.581,Z 314.868,A -85,B 0,C 180,E1 -7520.855,E2 -7520.855} C_VEL
LIN {X 0,Y 467.558,Z 314.865,A -85,B 0,C 180,E1 -7524.259,E2 -7524.259} C_VEL
LIN {X 0,Y 467.577,Z 314.865,A -85,B 0,C 180,E1 -7527.32,E2 -7527.32} C_VEL
LIN {X 0,Y 467.574,Z 314.868,A -85,B 0,C 180,E1 -7530.664,E2 -7530.664} C_VEL
LIN {X 0,Y 467.621,Z 314.859,A -85,B 0,C 180,E1 -7533.2,E2 -7533.2} C_VEL
LIN {X 0,Y 467.586,Z 314.865,A -85,B 0,C 180,E1 -7536.467,E2 -7536.467} C_VEL
LIN {X 0,Y 467.617,Z 314.857,A -85,B 0,C 180,E1 -7539.777,E2 -7539.777} C_VEL
LIN {X 0,Y 467.603,Z 314.865,A -85,B 0,C 180,E1 -7542.506,E2 -7542.506} C_VEL
LIN {X 0,Y 467.599,Z 314.861,A -85,B 0,C 180,E1 -7545.196,E2 -7545.196} C_VEL
LIN {X 0,Y 467.648,Z 314.854,A -85,B 0,C 180,E1 -7547.854,E2 -7547.854} C_VEL
LIN {X 0,Y 467.674,Z 314.85,A -85,B 0,C 180,E1 -7551.357,E2 -7551.357} C_VEL
LIN {X 0,Y 467.737,Z 314.844,A -85,B 0,C 180,E1 -7553.962,E2 -7553.962} C_VEL
LIN {X 0,Y 467.853,Z 314.827,A -85,B 0,C 180,E1 -7557.417,E2 -7557.417} C_VEL
LIN {X 0,Y 467.874,Z 314.828,A -85,B 0,C 180,E1 -7560,E2 -7560} C_VEL
LIN {X 0,Y 467.853,Z 314.832,A -85,B 0,C 180,E1 -7562.583,E2 -7562.583} C_VEL
LIN {X 0,Y 467.736,Z 314.847,A -85,B 0,C 180,E1 -7566.037,E2 -7566.037} C_VEL
LIN {X 0,Y 467.674,Z 314.853,A -85,B 0,C 180,E1 -7568.643,E2 -7568.643} C_VEL
LIN {X 0,Y 467.674,Z 314.858,A -85,B 0,C 180,E1 -7572.145,E2 -7572.145} C_VEL
LIN {X 0,Y 467.658,Z 314.857,A -85,B 0,C 180,E1 -7575.893,E2 -7575.893} C_VEL
LIN {X 0,Y 467.615,Z 314.858,A -85,B 0,C 180,E1 -7579.308,E2 -7579.308} C_VEL
LIN {X 0,Y 467.529,Z 314.876,A -85,B 0,C 180,E1 -7582.074,E2 -7582.074} C_VEL
LIN {X 0,Y 467.595,Z 314.86,A -85,B 0,C 180,E1 -7584.888,E2 -7584.888} C_VEL
LIN {X 0,Y 467.621,Z 314.862,A -85,B 0,C 180,E1 -7587.769,E2 -7587.769} C_VEL
LIN {X 0,Y 467.565,Z 314.863,A -85,B 0,C 180,E1 -7591.046,E2 -7591.046} C_VEL
LIN {X 0,Y 467.583,Z 314.864,A -85,B 0,C 180,E1 -7594.243,E2 -7594.243} C_VEL
LIN {X 0,Y 467.545,Z 314.869,A -85,B 0,C 180,E1 -7597.188,E2 -7597.188} C_VEL
LIN {X 0,Y 467.59,Z 314.866,A -85,B 0,C 180,E1 -7600.263,E2 -7600.263} C_VEL
LIN {X 0,Y 467.58,Z 314.867,A -85,B 0,C 180,E1 -7602.568,E2 -7602.568} C_VEL
LIN {X 0,Y 467.623,Z 315.046,A -85,B 0,C 180,E1 -7605.422,E2 -7605.422} C_VEL
LIN {X 0,Y 469.992,Z 326.258,A -85,B 0,C 180,E1 -7608.858,E2 -7608.858} C_VEL
LIN {X 0,Y 471.001,Z 332.01,A -85,B 0,C 180,E1 -7610.534,E2 -7610.534} C_VEL
LIN {X 0,Y 470.947,Z 336.406,A -85,B 0,C 180,E1 -7611.736,E2 -7611.736} C_VEL
LIN {X 0,Y 470.032,Z 350.284,A -85,B 0,C 180,E1 -7615.378,E2 -7615.378} C_VEL
LIN {X 0,Y 469.307,Z 364.483,A -85,B 0,C 180,E1 -7618.989,E2 -7618.989} C_VEL
LIN {X 0,Y 468.802,Z 375.906,A -85,B 0,C 180,E1 -7621.815,E2 -7621.815} C_VEL
LIN {X 0,Y 468.334,Z 389.706,A -85,B 0,C 180,E1 -7625.155,E2 -7625.155} C_VEL
LIN {X 0,Y 467.941,Z 401.471,A -85,B 0,C 180,E1 -7627.947,E2 -7627.947} C_VEL
LIN {X 0,Y 467.578,Z 415.627,A -85,B 0,C 180,E1 -7631.25,E2 -7631.25} C_VEL
LIN {X 0,Y 467.581,Z 416.775,A -85,B 0,C 180,E1 -7631.395,E2 -7631.395} C_VEL
LIN {X 0,Y 469.901,Z 433.749,A -85,B 0,C 180,E1 -7631.907,E2 -7631.907} C_VEL
LIN {X 0,Y 471.166,Z 443.895,A -85,B 0,C 180,E1 -7632.308,E2 -7632.308} C_VEL
LIN {X 0,Y 470.597,Z 457.148,A -85,B 0,C 180,E1 -7632.899,E2 -7632.899} C_VEL
LIN {X 0,Y 470.029,Z 469.466,A -85,B 0,C 180,E1 -7633.608,E2 -7633.608} C_VEL
LIN {X 0,Y 469.263,Z 483.032,A -85,B 0,C 180,E1 -7634.584,E2 -7634.584} C_VEL
LIN {X 0,Y 468.667,Z 495.178,A -85,B 0,C 180,E1 -7635.675,E2 -7635.675} C_VEL
LIN {X 0,Y 468.129,Z 505.28,A -85,B 0,C 180,E1 -7636.766,E2 -7636.766} C_VEL
LIN {X 0,Y 467.702,Z 515.388,A -85,B 0,C 180,E1 -7638.077,E2 -7638.077} C_VEL
LIN {X 0,Y 467.313,Z 525.054,A -85,B 0,C 180,E1 -7639.604,E2 -7639.604} C_VEL
LIN {X 0,Y 467.06,Z 532.881,A -85,B 0,C 180,E1 -7641.128,E2 -7641.128} C_VEL
LIN {X 0,Y 466.936,Z 539.151,A -85,B 0,C 180,E1 -7642.651,E2 -7642.651} C_VEL
LIN {X 0,Y 466.945,Z 544.661,A -85,B 0,C 180,E1 -7644.387,E2 -7644.387} C_VEL
LIN {X 0,Y 466.937,Z 547.692,A -85,B 0,C 180,E1 -7645.685,E2 -7645.685} C_VEL
LIN {X 0,Y 466.94,Z 550.455,A -85,B 0,C 180,E1 -7647.413,E2 -7647.413} C_VEL
LIN {X 0,Y 466.896,Z 551.766,A -85,B 0,C 180,E1 -7649.138,E2 -7649.138} C_VEL
LIN {X 0,Y 467.015,Z 551.907,A -85,B 0,C 180,E1 -7650.001,E2 -7650.001} C_VEL
LIN {X 0,Y 467.033,Z 551.675,A -85,B 0,C 180,E1 -7650.863,E2 -7650.863} C_VEL
LIN {X 0,Y 466.981,Z 550.12,A -85,B 0,C 180,E1 -7652.589,E2 -7652.589} C_VEL
LIN {X 0,Y 467.071,Z 547.112,A -85,B 0,C 180,E1 -7654.315,E2 -7654.315} C_VEL
LIN {X 0,Y 467.042,Z 543.847,A -85,B 0,C 180,E1 -7655.614,E2 -7655.614} C_VEL
LIN {X 0,Y 467.035,Z 539.625,A -85,B 0,C 180,E1 -7656.915,E2 -7656.915} C_VEL
LIN {X 0,Y 467.119,Z 534.435,A -85,B 0,C 180,E1 -7658.218,E2 -7658.218} C_VEL
LIN {X 0,Y 467.231,Z 526.941,A -85,B 0,C 180,E1 -7659.743,E2 -7659.743} C_VEL
LIN {X 0,Y 467.491,Z 517.681,A -85,B 0,C 180,E1 -7661.271,E2 -7661.271} C_VEL
LIN {X 0,Y 467.887,Z 507.662,A -85,B 0,C 180,E1 -7662.632,E2 -7662.632} C_VEL
LIN {X 0,Y 468.311,Z 496.463,A -85,B 0,C 180,E1 -7663.894,E2 -7663.894} C_VEL
LIN {X 0,Y 468.908,Z 484.77,A -85,B 0,C 180,E1 -7664.984,E2 -7664.984} C_VEL
LIN {X 0,Y 469.514,Z 472.002,A -85,B 0,C 180,E1 -7665.966,E2 -7665.966} C_VEL
LIN {X 0,Y 470.176,Z 458.988,A -85,B 0,C 180,E1 -7666.776,E2 -7666.776} C_VEL
LIN {X 0,Y 470.815,Z 444.602,A -85,B 0,C 180,E1 -7667.483,E2 -7667.483} C_VEL
LIN {X 0,Y 470.34,Z 439.185,A -85,B 0,C 180,E1 -7667.726,E2 -7667.726} C_VEL
LIN {X 0,Y 469.138,Z 426.989,A -85,B 0,C 180,E1 -7668.196,E2 -7668.196} C_VEL
LIN {X 0,Y 467.419,Z 410.893,A -85,B 0,C 180,E1 -7668.692,E2 -7668.692} C_VEL
LIN {X 0,Y 467.529,Z 405.617,A -85,B 0,C 180,E1 -7669.769,E2 -7669.769} C_VEL
LIN {X 0,Y 467.685,Z 390.764,A -85,B 0,C 180,E1 -7672.999,E2 -7672.999} C_VEL
LIN {X 0,Y 467.837,Z 375.831,A -85,B 0,C 180,E1 -7676.306,E2 -7676.306} C_VEL
LIN {X 0,Y 468.059,Z 362.113,A -85,B 0,C 180,E1 -7679.439,E2 -7679.439} C_VEL
LIN {X 0,Y 468.177,Z 350.507,A -85,B 0,C 180,E1 -7682.203,E2 -7682.203} C_VEL
LIN {X 0,Y 468.77,Z 335.758,A -85,B 0,C 180,E1 -7685.944,E2 -7685.944} C_VEL
LIN {X 0,Y 469.591,Z 326.941,A -85,B 0,C 180,E1 -7688.37,E2 -7688.37} C_VEL
LIN {X 0,Y 469.241,Z 323.188,A -85,B 0,C 180,E1 -7689.535,E2 -7689.535} C_VEL
LIN {X 0,Y 467.731,Z 315.545,A -85,B 0,C 180,E1 -7692.268,E2 -7692.268} C_VEL
LIN {X 0,Y 467.589,Z 314.916,A -85,B 0,C 180,E1 -7692.567,E2 -7692.567} C_VEL
LIN {X 0,Y 467.574,Z 314.87,A -85,B 0,C 180,E1 -7695.054,E2 -7695.054} C_VEL
LIN {X 0,Y 467.592,Z 314.869,A -85,B 0,C 180,E1 -7697.44,E2 -7697.44} C_VEL
LIN {X 0,Y 467.619,Z 314.862,A -85,B 0,C 180,E1 -7700.859,E2 -7700.859} C_VEL
LIN {X 0,Y 467.567,Z 314.866,A -85,B 0,C 180,E1 -7704.261,E2 -7704.261} C_VEL
LIN {X 0,Y 467.585,Z 314.867,A -85,B 0,C 180,E1 -7707.321,E2 -7707.321} C_VEL
LIN {X 0,Y 467.573,Z 314.866,A -85,B 0,C 180,E1 -7710.668,E2 -7710.668} C_VEL
LIN {X 0,Y 467.62,Z 314.863,A -85,B 0,C 180,E1 -7713.2,E2 -7713.2} C_VEL
LIN {X 0,Y 467.596,Z 314.864,A -85,B 0,C 180,E1 -7716.468,E2 -7716.468} C_VEL
